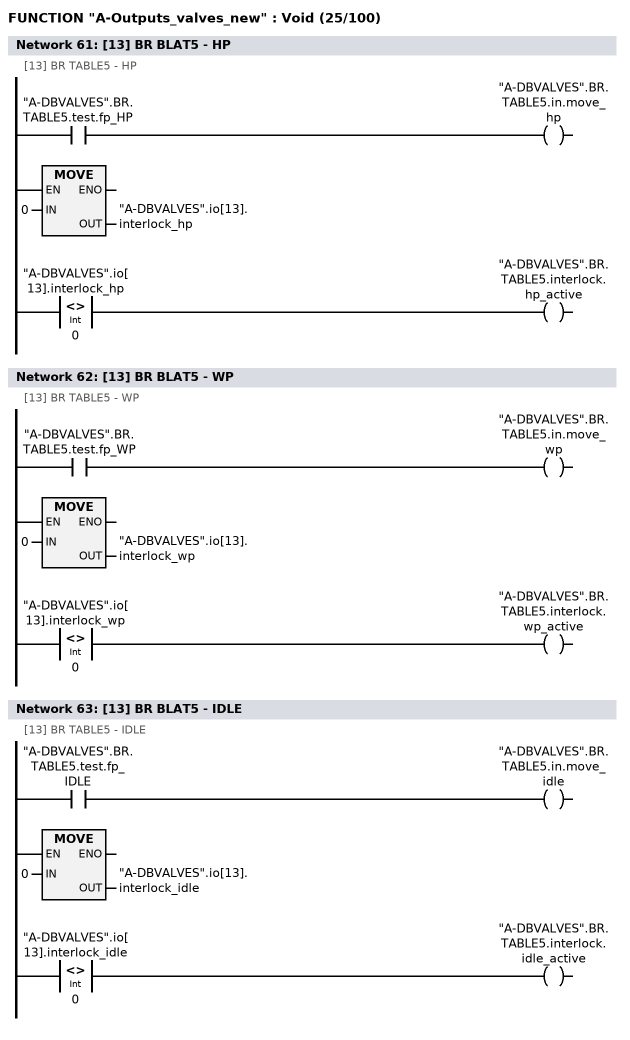
      O "A-DBVALVES".BR.TABLE5.test.fp_HP;
//    O     "A-Flags".STATION.IN_HP_STEP
      = "A-DBVALVES".BR.TABLE5.in.move_hp;

// Interlock hp
      L 0;
      T "A-DBVALVES".io[13].interlock_hp;

//{INTERLOCK_HP13}

      A(;
      L "A-DBVALVES".io[13].interlock_hp;
      L 0;
      <>I;
      );
      = "A-DBVALVES".BR.TABLE5.interlock.hp_active;
NETWORK
TITLE = [13] BR BLAT5 - WP
//[13] BR TABLE5 - WP
      O "A-DBVALVES".BR.TABLE5.test.fp_WP;
      = "A-DBVALVES".BR.TABLE5.in.move_wp;

// Interlock wp
      L 0;
      T "A-DBVALVES".io[13].interlock_wp;

//{INTERLOCK_WP13}

      A(;
      L "A-DBVALVES".io[13].interlock_wp;
      L 0;
      <>I;
      );
      = "A-DBVALVES".BR.TABLE5.interlock.wp_active;
NETWORK
TITLE = [13] BR BLAT5 - IDLE
//[13] BR TABLE5 - IDLE
      O "A-DBVALVES".BR.TABLE5.test.fp_IDLE;
      = "A-DBVALVES".BR.TABLE5.in.move_idle;

// Interlock idle
      L 0;
      T "A-DBVALVES".io[13].interlock_idle;

//{INTERLOCK_IDLE13}

      A(;
      L "A-DBVALVES".io[13].interlock_idle;
      L 0;
      <>I;
      );
      = "A-DBVALVES".BR.TABLE5.interlock.idle_active;
NETWORK
TITLE = [13] BR BLAT5
//[13] BR TABLE5
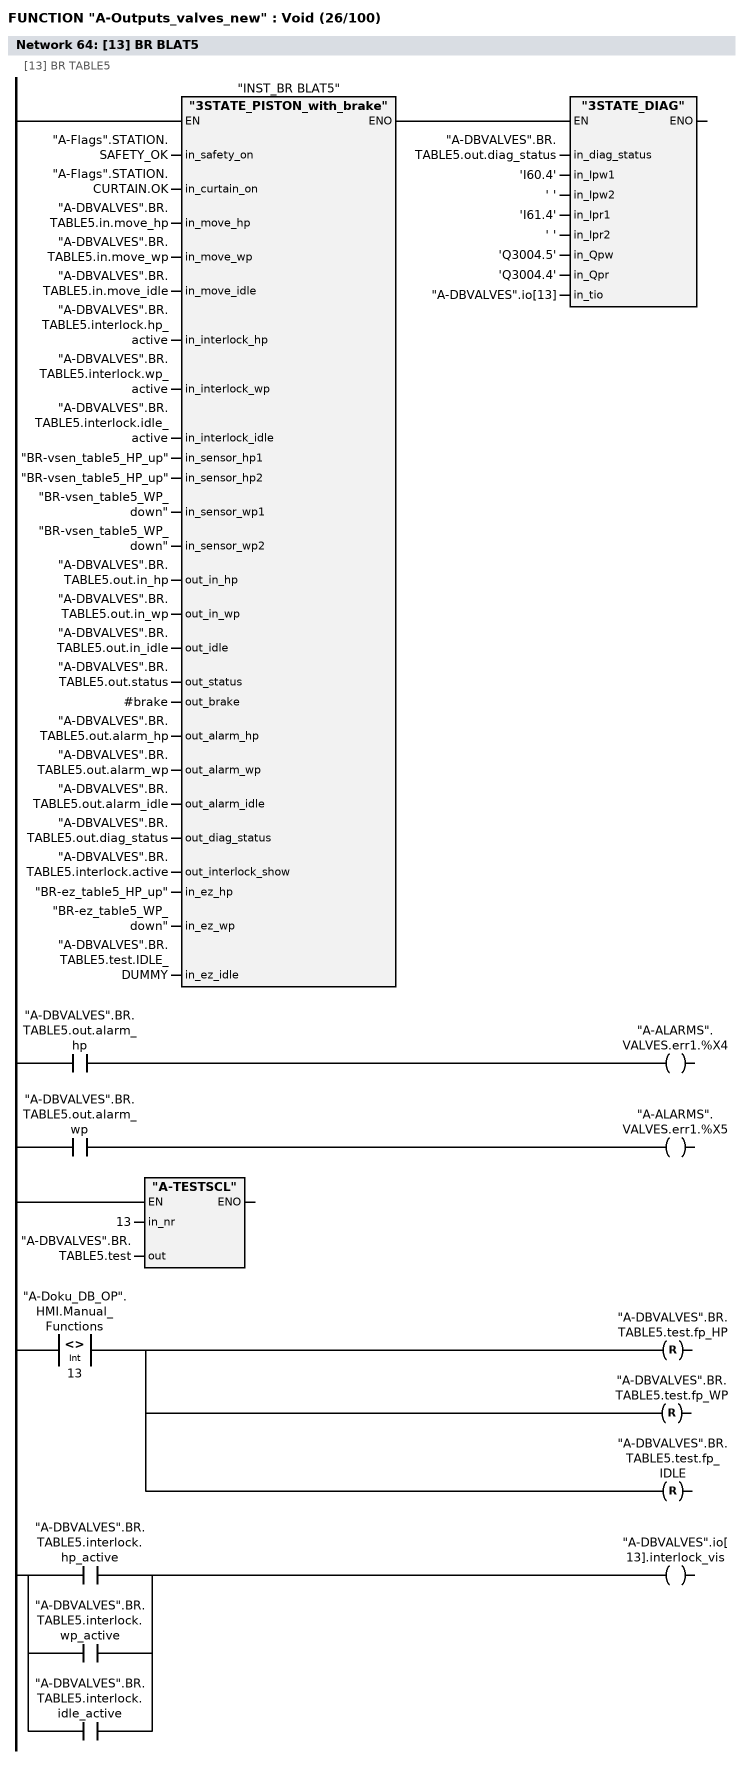
      CALL "3STATE_PISTON_with_brake", "INST_BR BLAT5"
      (  in_safety_on                := "A-Flags".STATION.SAFETY_OK ,
         in_curtain_on               := "A-Flags".STATION.CURTAIN.OK ,
         in_move_hp                  := "A-DBVALVES".BR.TABLE5.in.move_hp ,
         in_move_wp                  := "A-DBVALVES".BR.TABLE5.in.move_wp ,
         in_move_idle                := "A-DBVALVES".BR.TABLE5.in.move_idle ,
         in_interlock_hp             := "A-DBVALVES".BR.TABLE5.interlock.hp_active ,
         in_interlock_wp             := "A-DBVALVES".BR.TABLE5.interlock.wp_active ,
         in_interlock_idle           := "A-DBVALVES".BR.TABLE5.interlock.idle_active ,
         in_sensor_hp1               := "BR-vsen_table5_HP_up" ,
         in_sensor_hp2               := "BR-vsen_table5_HP_up" ,
         in_sensor_wp1               := "BR-vsen_table5_WP_down" ,
         in_sensor_wp2               := "BR-vsen_table5_WP_down" ,
         out_in_hp                   := "A-DBVALVES".BR.TABLE5.out.in_hp ,
         out_in_wp                   := "A-DBVALVES".BR.TABLE5.out.in_wp ,
         out_idle                    := "A-DBVALVES".BR.TABLE5.out.in_idle ,
         out_status                  := "A-DBVALVES".BR.TABLE5.out.status ,
         out_brake                   := #brake ,
         out_alarm_hp                := "A-DBVALVES".BR.TABLE5.out.alarm_hp ,
         out_alarm_wp                := "A-DBVALVES".BR.TABLE5.out.alarm_wp ,
         out_alarm_idle              := "A-DBVALVES".BR.TABLE5.out.alarm_idle ,
         out_diag_status             := "A-DBVALVES".BR.TABLE5.out.diag_status ,
         out_interlock_show          := "A-DBVALVES".BR.TABLE5.interlock.active ,
         in_ez_hp                    := "BR-ez_table5_HP_up" ,
         in_ez_wp                    := "BR-ez_table5_WP_down" ,
         in_ez_idle                  := "A-DBVALVES".BR.TABLE5.test.IDLE_DUMMY
      );

      CALL "3STATE_DIAG"
      (  in_diag_status              := "A-DBVALVES".BR.TABLE5.out.diag_status ,
         in_Ipw1                     := 'I60.4' ,
         in_Ipw2                     := ' ' ,
         in_Ipr1                     := 'I61.4' ,
         in_Ipr2                     := ' ' ,
         in_Qpw                      := 'Q3004.5' ,
         in_Qpr                      := 'Q3004.4' ,
         in_tio                      := "A-DBVALVES".io[13]
      );

      A "A-DBVALVES".BR.TABLE5.out.alarm_hp;
      = "A-ALARMS".VALVES.err1.%X4;

      A "A-DBVALVES".BR.TABLE5.out.alarm_wp;
      = "A-ALARMS".VALVES.err1.%X5;

      CALL "A-TESTSCL"
      (  in_nr                       := 13 ,
         out                         := "A-DBVALVES".BR.TABLE5.test
      );

      A(;
      L "A-Doku_DB_OP".HMI.Manual_Functions;
      L 13;
      <>I;
      );
      R "A-DBVALVES".BR.TABLE5.test.fp_HP;
      R "A-DBVALVES".BR.TABLE5.test.fp_WP;
      R "A-DBVALVES".BR.TABLE5.test.fp_IDLE;

      O "A-DBVALVES".BR.TABLE5.interlock.hp_active;
      O "A-DBVALVES".BR.TABLE5.interlock.wp_active;
      O "A-DBVALVES".BR.TABLE5.interlock.idle_active;
      = "A-DBVALVES".io[13].interlock_vis;
NETWORK
TITLE = -

NETWORK
TITLE = [14] BR BLAT_LEWY - HP
//[14] BR TABLE_LEFT - HP
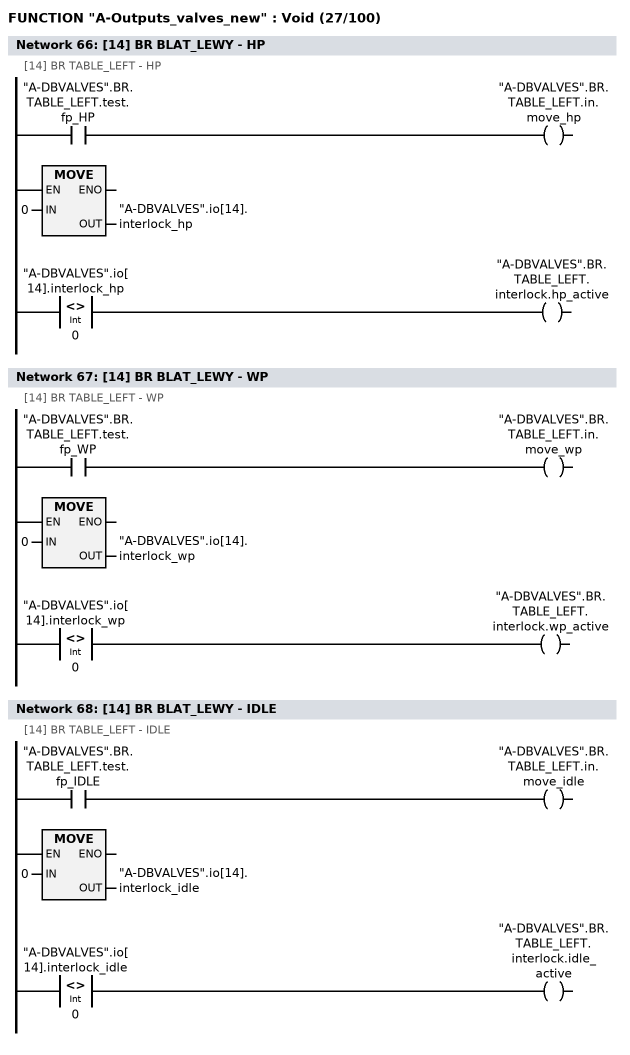
      O "A-DBVALVES".BR.TABLE_LEFT.test.fp_HP;
//    O     "A-Flags".STATION.IN_HP_STEP
      = "A-DBVALVES".BR.TABLE_LEFT.in.move_hp;

// Interlock hp
      L 0;
      T "A-DBVALVES".io[14].interlock_hp;

//{INTERLOCK_HP14}

      A(;
      L "A-DBVALVES".io[14].interlock_hp;
      L 0;
      <>I;
      );
      = "A-DBVALVES".BR.TABLE_LEFT.interlock.hp_active;
NETWORK
TITLE = [14] BR BLAT_LEWY - WP
//[14] BR TABLE_LEFT - WP
      O "A-DBVALVES".BR.TABLE_LEFT.test.fp_WP;
      = "A-DBVALVES".BR.TABLE_LEFT.in.move_wp;

// Interlock wp
      L 0;
      T "A-DBVALVES".io[14].interlock_wp;

//{INTERLOCK_WP14}

      A(;
      L "A-DBVALVES".io[14].interlock_wp;
      L 0;
      <>I;
      );
      = "A-DBVALVES".BR.TABLE_LEFT.interlock.wp_active;
NETWORK
TITLE = [14] BR BLAT_LEWY - IDLE
//[14] BR TABLE_LEFT - IDLE
      O "A-DBVALVES".BR.TABLE_LEFT.test.fp_IDLE;
      = "A-DBVALVES".BR.TABLE_LEFT.in.move_idle;

// Interlock idle
      L 0;
      T "A-DBVALVES".io[14].interlock_idle;

//{INTERLOCK_IDLE14}

      A(;
      L "A-DBVALVES".io[14].interlock_idle;
      L 0;
      <>I;
      );
      = "A-DBVALVES".BR.TABLE_LEFT.interlock.idle_active;
NETWORK
TITLE = [14] BR BLAT_LEWY
//[14] BR TABLE_LEFT
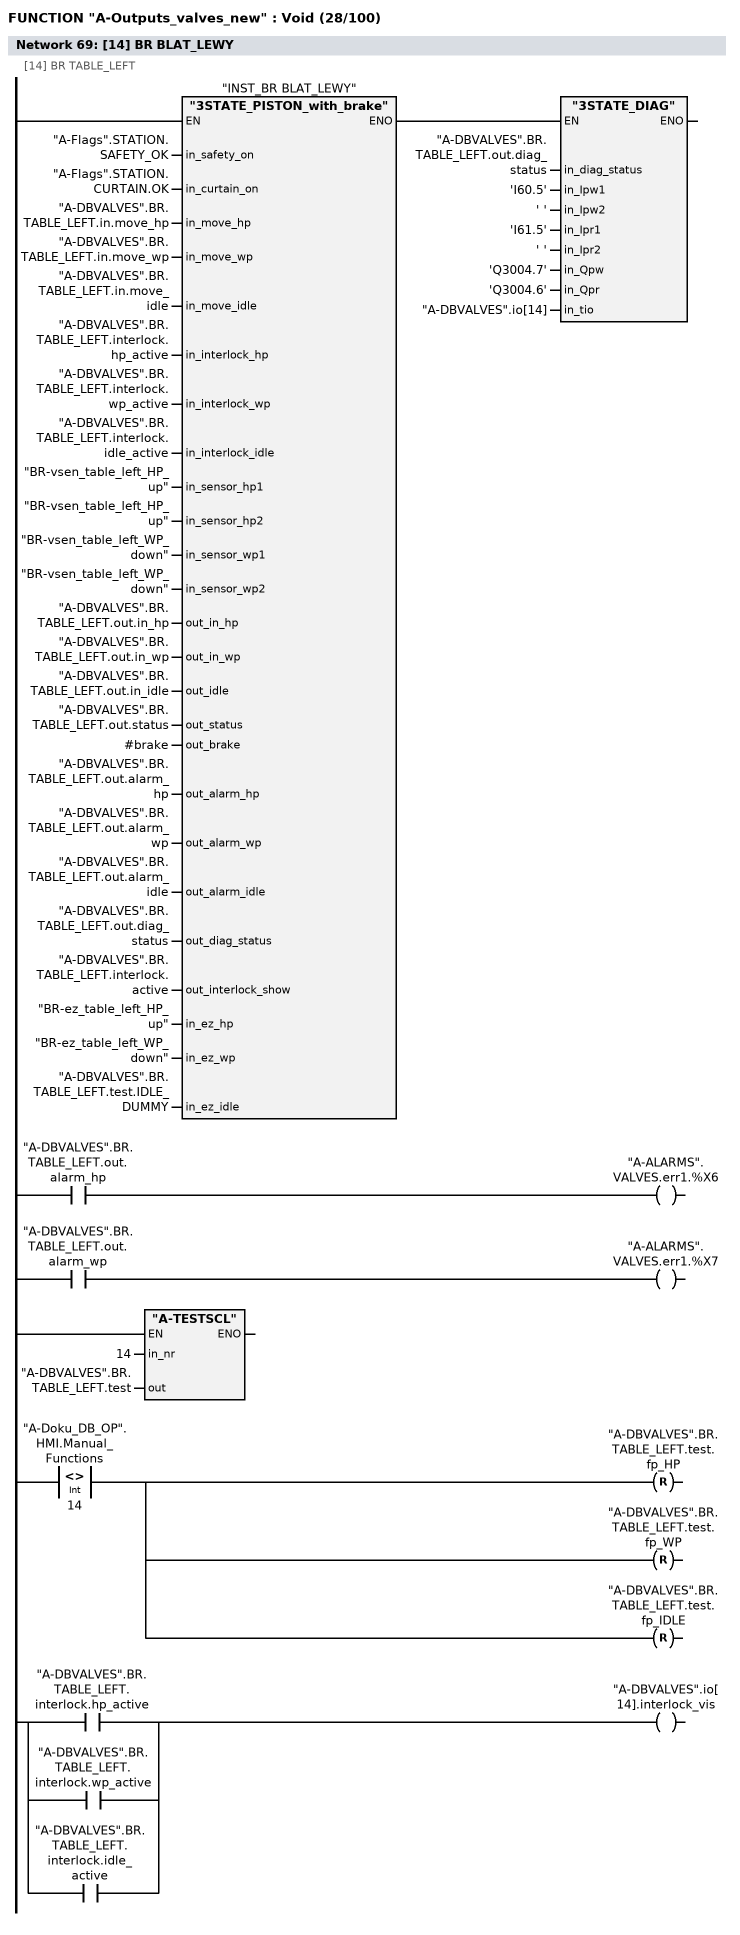
      CALL "3STATE_PISTON_with_brake", "INST_BR BLAT_LEWY"
      (  in_safety_on                := "A-Flags".STATION.SAFETY_OK ,
         in_curtain_on               := "A-Flags".STATION.CURTAIN.OK ,
         in_move_hp                  := "A-DBVALVES".BR.TABLE_LEFT.in.move_hp ,
         in_move_wp                  := "A-DBVALVES".BR.TABLE_LEFT.in.move_wp ,
         in_move_idle                := "A-DBVALVES".BR.TABLE_LEFT.in.move_idle ,
         in_interlock_hp             := "A-DBVALVES".BR.TABLE_LEFT.interlock.hp_active ,
         in_interlock_wp             := "A-DBVALVES".BR.TABLE_LEFT.interlock.wp_active ,
         in_interlock_idle           := "A-DBVALVES".BR.TABLE_LEFT.interlock.idle_active ,
         in_sensor_hp1               := "BR-vsen_table_left_HP_up" ,
         in_sensor_hp2               := "BR-vsen_table_left_HP_up" ,
         in_sensor_wp1               := "BR-vsen_table_left_WP_down" ,
         in_sensor_wp2               := "BR-vsen_table_left_WP_down" ,
         out_in_hp                   := "A-DBVALVES".BR.TABLE_LEFT.out.in_hp ,
         out_in_wp                   := "A-DBVALVES".BR.TABLE_LEFT.out.in_wp ,
         out_idle                    := "A-DBVALVES".BR.TABLE_LEFT.out.in_idle ,
         out_status                  := "A-DBVALVES".BR.TABLE_LEFT.out.status ,
         out_brake                   := #brake ,
         out_alarm_hp                := "A-DBVALVES".BR.TABLE_LEFT.out.alarm_hp ,
         out_alarm_wp                := "A-DBVALVES".BR.TABLE_LEFT.out.alarm_wp ,
         out_alarm_idle              := "A-DBVALVES".BR.TABLE_LEFT.out.alarm_idle ,
         out_diag_status             := "A-DBVALVES".BR.TABLE_LEFT.out.diag_status ,
         out_interlock_show          := "A-DBVALVES".BR.TABLE_LEFT.interlock.active ,
         in_ez_hp                    := "BR-ez_table_left_HP_up" ,
         in_ez_wp                    := "BR-ez_table_left_WP_down" ,
         in_ez_idle                  := "A-DBVALVES".BR.TABLE_LEFT.test.IDLE_DUMMY
      );

      CALL "3STATE_DIAG"
      (  in_diag_status              := "A-DBVALVES".BR.TABLE_LEFT.out.diag_status ,
         in_Ipw1                     := 'I60.5' ,
         in_Ipw2                     := ' ' ,
         in_Ipr1                     := 'I61.5' ,
         in_Ipr2                     := ' ' ,
         in_Qpw                      := 'Q3004.7' ,
         in_Qpr                      := 'Q3004.6' ,
         in_tio                      := "A-DBVALVES".io[14]
      );

      A "A-DBVALVES".BR.TABLE_LEFT.out.alarm_hp;
      = "A-ALARMS".VALVES.err1.%X6;

      A "A-DBVALVES".BR.TABLE_LEFT.out.alarm_wp;
      = "A-ALARMS".VALVES.err1.%X7;

      CALL "A-TESTSCL"
      (  in_nr                       := 14 ,
         out                         := "A-DBVALVES".BR.TABLE_LEFT.test
      );

      A(;
      L "A-Doku_DB_OP".HMI.Manual_Functions;
      L 14;
      <>I;
      );
      R "A-DBVALVES".BR.TABLE_LEFT.test.fp_HP;
      R "A-DBVALVES".BR.TABLE_LEFT.test.fp_WP;
      R "A-DBVALVES".BR.TABLE_LEFT.test.fp_IDLE;

      O "A-DBVALVES".BR.TABLE_LEFT.interlock.hp_active;
      O "A-DBVALVES".BR.TABLE_LEFT.interlock.wp_active;
      O "A-DBVALVES".BR.TABLE_LEFT.interlock.idle_active;
      = "A-DBVALVES".io[14].interlock_vis;
NETWORK
TITLE = -

NETWORK
TITLE = [15] BR BLAT_PRAWY - HP
//[15] BR TABLE_RIGHT - HP
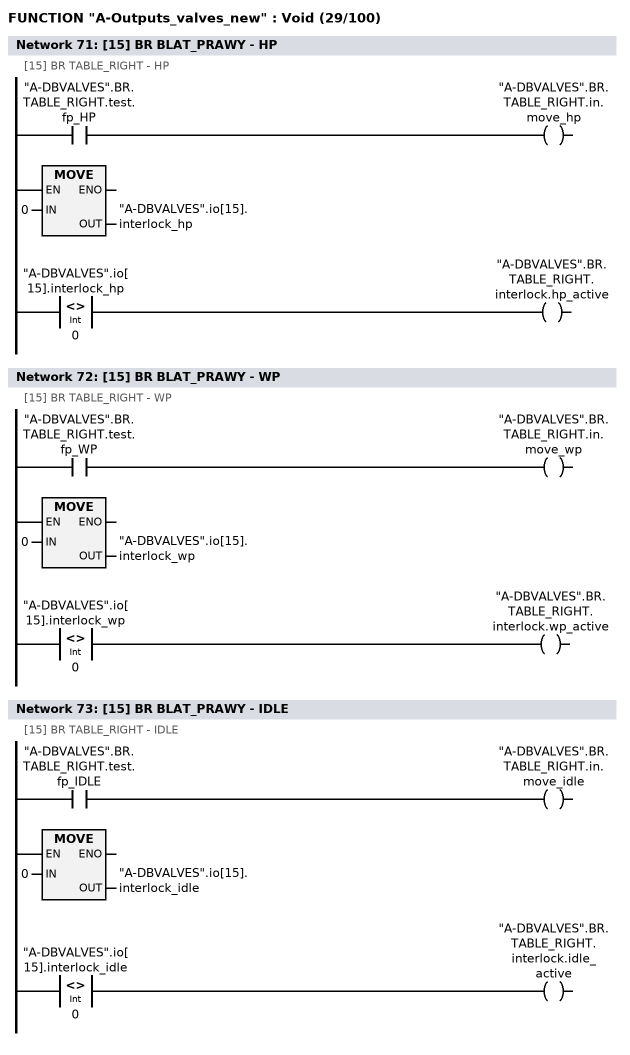
      O "A-DBVALVES".BR.TABLE_RIGHT.test.fp_HP;
//    O     "A-Flags".STATION.IN_HP_STEP
      = "A-DBVALVES".BR.TABLE_RIGHT.in.move_hp;

// Interlock hp
      L 0;
      T "A-DBVALVES".io[15].interlock_hp;

//{INTERLOCK_HP15}

      A(;
      L "A-DBVALVES".io[15].interlock_hp;
      L 0;
      <>I;
      );
      = "A-DBVALVES".BR.TABLE_RIGHT.interlock.hp_active;
NETWORK
TITLE = [15] BR BLAT_PRAWY - WP
//[15] BR TABLE_RIGHT - WP
      O "A-DBVALVES".BR.TABLE_RIGHT.test.fp_WP;
      = "A-DBVALVES".BR.TABLE_RIGHT.in.move_wp;

// Interlock wp
      L 0;
      T "A-DBVALVES".io[15].interlock_wp;

//{INTERLOCK_WP15}

      A(;
      L "A-DBVALVES".io[15].interlock_wp;
      L 0;
      <>I;
      );
      = "A-DBVALVES".BR.TABLE_RIGHT.interlock.wp_active;
NETWORK
TITLE = [15] BR BLAT_PRAWY - IDLE
//[15] BR TABLE_RIGHT - IDLE
      O "A-DBVALVES".BR.TABLE_RIGHT.test.fp_IDLE;
      = "A-DBVALVES".BR.TABLE_RIGHT.in.move_idle;

// Interlock idle
      L 0;
      T "A-DBVALVES".io[15].interlock_idle;

//{INTERLOCK_IDLE15}

      A(;
      L "A-DBVALVES".io[15].interlock_idle;
      L 0;
      <>I;
      );
      = "A-DBVALVES".BR.TABLE_RIGHT.interlock.idle_active;
NETWORK
TITLE = [15] BR BLAT_PRAWY
//[15] BR TABLE_RIGHT
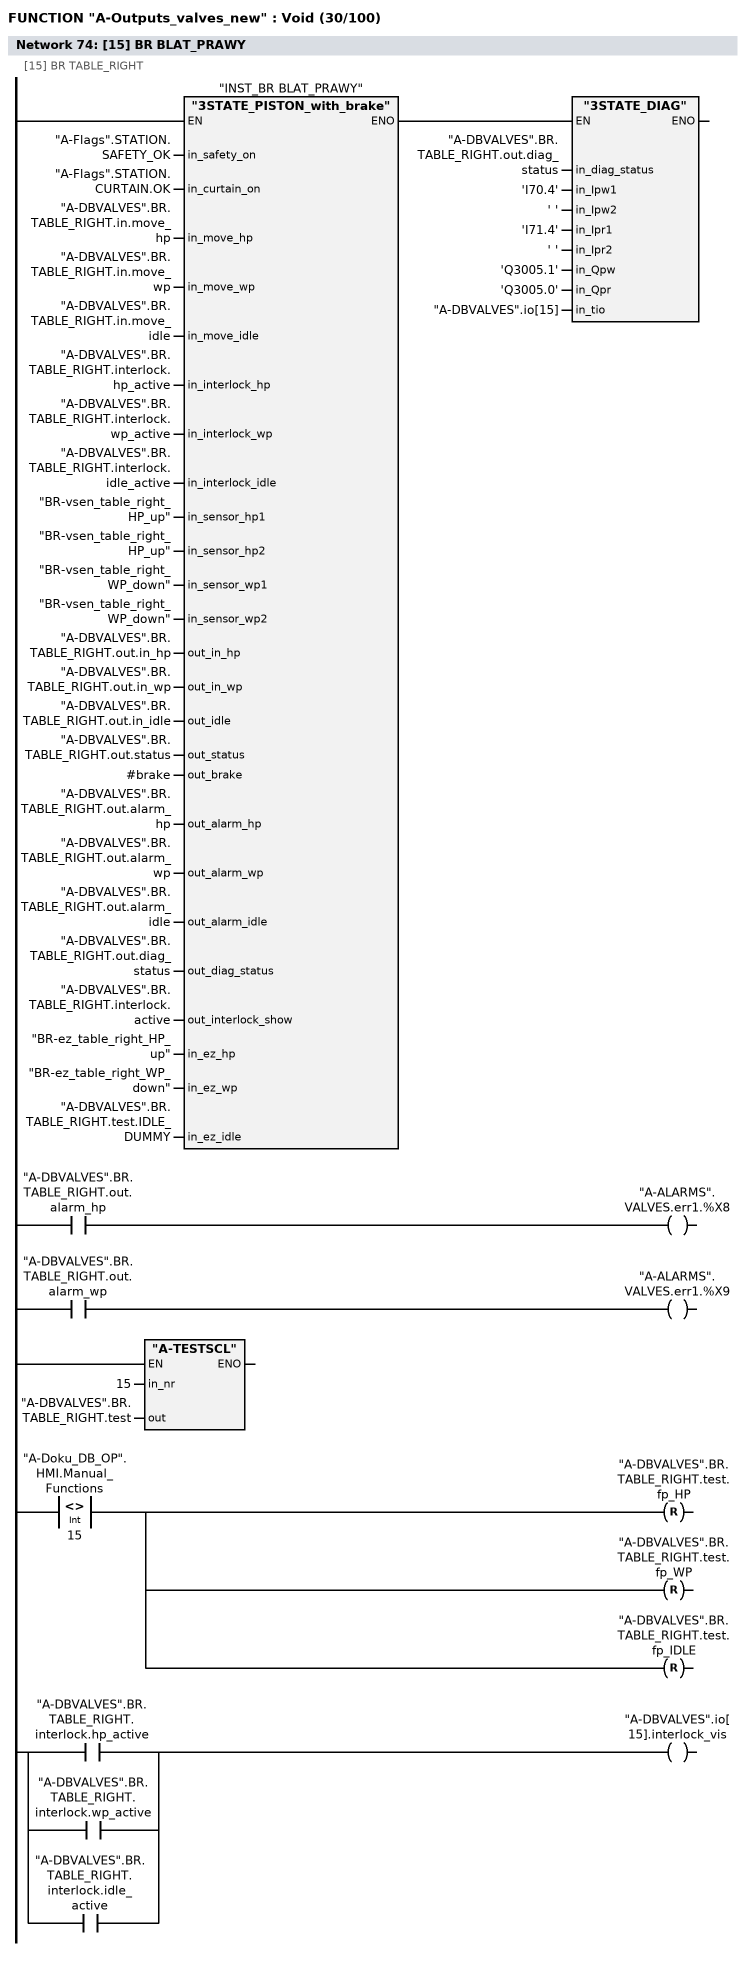
      CALL "3STATE_PISTON_with_brake", "INST_BR BLAT_PRAWY"
      (  in_safety_on                := "A-Flags".STATION.SAFETY_OK ,
         in_curtain_on               := "A-Flags".STATION.CURTAIN.OK ,
         in_move_hp                  := "A-DBVALVES".BR.TABLE_RIGHT.in.move_hp ,
         in_move_wp                  := "A-DBVALVES".BR.TABLE_RIGHT.in.move_wp ,
         in_move_idle                := "A-DBVALVES".BR.TABLE_RIGHT.in.move_idle ,
         in_interlock_hp             := "A-DBVALVES".BR.TABLE_RIGHT.interlock.hp_active ,
         in_interlock_wp             := "A-DBVALVES".BR.TABLE_RIGHT.interlock.wp_active ,
         in_interlock_idle           := "A-DBVALVES".BR.TABLE_RIGHT.interlock.idle_active ,
         in_sensor_hp1               := "BR-vsen_table_right_HP_up" ,
         in_sensor_hp2               := "BR-vsen_table_right_HP_up" ,
         in_sensor_wp1               := "BR-vsen_table_right_WP_down" ,
         in_sensor_wp2               := "BR-vsen_table_right_WP_down" ,
         out_in_hp                   := "A-DBVALVES".BR.TABLE_RIGHT.out.in_hp ,
         out_in_wp                   := "A-DBVALVES".BR.TABLE_RIGHT.out.in_wp ,
         out_idle                    := "A-DBVALVES".BR.TABLE_RIGHT.out.in_idle ,
         out_status                  := "A-DBVALVES".BR.TABLE_RIGHT.out.status ,
         out_brake                   := #brake ,
         out_alarm_hp                := "A-DBVALVES".BR.TABLE_RIGHT.out.alarm_hp ,
         out_alarm_wp                := "A-DBVALVES".BR.TABLE_RIGHT.out.alarm_wp ,
         out_alarm_idle              := "A-DBVALVES".BR.TABLE_RIGHT.out.alarm_idle ,
         out_diag_status             := "A-DBVALVES".BR.TABLE_RIGHT.out.diag_status ,
         out_interlock_show          := "A-DBVALVES".BR.TABLE_RIGHT.interlock.active ,
         in_ez_hp                    := "BR-ez_table_right_HP_up" ,
         in_ez_wp                    := "BR-ez_table_right_WP_down" ,
         in_ez_idle                  := "A-DBVALVES".BR.TABLE_RIGHT.test.IDLE_DUMMY
      );

      CALL "3STATE_DIAG"
      (  in_diag_status              := "A-DBVALVES".BR.TABLE_RIGHT.out.diag_status ,
         in_Ipw1                     := 'I70.4' ,
         in_Ipw2                     := ' ' ,
         in_Ipr1                     := 'I71.4' ,
         in_Ipr2                     := ' ' ,
         in_Qpw                      := 'Q3005.1' ,
         in_Qpr                      := 'Q3005.0' ,
         in_tio                      := "A-DBVALVES".io[15]
      );

      A "A-DBVALVES".BR.TABLE_RIGHT.out.alarm_hp;
      = "A-ALARMS".VALVES.err1.%X8;

      A "A-DBVALVES".BR.TABLE_RIGHT.out.alarm_wp;
      = "A-ALARMS".VALVES.err1.%X9;

      CALL "A-TESTSCL"
      (  in_nr                       := 15 ,
         out                         := "A-DBVALVES".BR.TABLE_RIGHT.test
      );

      A(;
      L "A-Doku_DB_OP".HMI.Manual_Functions;
      L 15;
      <>I;
      );
      R "A-DBVALVES".BR.TABLE_RIGHT.test.fp_HP;
      R "A-DBVALVES".BR.TABLE_RIGHT.test.fp_WP;
      R "A-DBVALVES".BR.TABLE_RIGHT.test.fp_IDLE;

      O "A-DBVALVES".BR.TABLE_RIGHT.interlock.hp_active;
      O "A-DBVALVES".BR.TABLE_RIGHT.interlock.wp_active;
      O "A-DBVALVES".BR.TABLE_RIGHT.interlock.idle_active;
      = "A-DBVALVES".io[15].interlock_vis;
NETWORK
TITLE = -

NETWORK
TITLE = [16] ST1 STACJA_PRZESUW - HP
//[16] ST1 STATION_MOVEMENT - HP
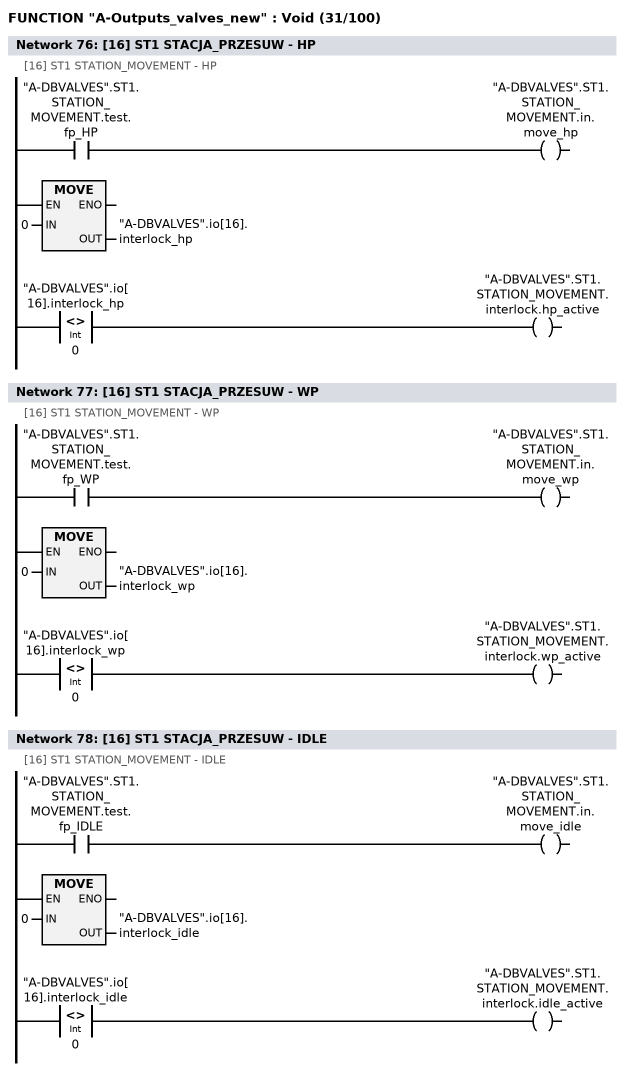
      O "A-DBVALVES".ST1.STATION_MOVEMENT.test.fp_HP;
//    O     "A-Flags".STATION.IN_HP_STEP
      = "A-DBVALVES".ST1.STATION_MOVEMENT.in.move_hp;

// Interlock hp
      L 0;
      T "A-DBVALVES".io[16].interlock_hp;

//{INTERLOCK_HP16}

      A(;
      L "A-DBVALVES".io[16].interlock_hp;
      L 0;
      <>I;
      );
      = "A-DBVALVES".ST1.STATION_MOVEMENT.interlock.hp_active;
NETWORK
TITLE = [16] ST1 STACJA_PRZESUW - WP
//[16] ST1 STATION_MOVEMENT - WP
      O "A-DBVALVES".ST1.STATION_MOVEMENT.test.fp_WP;
      = "A-DBVALVES".ST1.STATION_MOVEMENT.in.move_wp;

// Interlock wp
      L 0;
      T "A-DBVALVES".io[16].interlock_wp;

//{INTERLOCK_WP16}

      A(;
      L "A-DBVALVES".io[16].interlock_wp;
      L 0;
      <>I;
      );
      = "A-DBVALVES".ST1.STATION_MOVEMENT.interlock.wp_active;
NETWORK
TITLE = [16] ST1 STACJA_PRZESUW - IDLE
//[16] ST1 STATION_MOVEMENT - IDLE
      O "A-DBVALVES".ST1.STATION_MOVEMENT.test.fp_IDLE;
      = "A-DBVALVES".ST1.STATION_MOVEMENT.in.move_idle;

// Interlock idle
      L 0;
      T "A-DBVALVES".io[16].interlock_idle;

//{INTERLOCK_IDLE16}

      A(;
      L "A-DBVALVES".io[16].interlock_idle;
      L 0;
      <>I;
      );
      = "A-DBVALVES".ST1.STATION_MOVEMENT.interlock.idle_active;
NETWORK
TITLE = [16] ST1 STACJA_PRZESUW
//[16] ST1 STATION_MOVEMENT
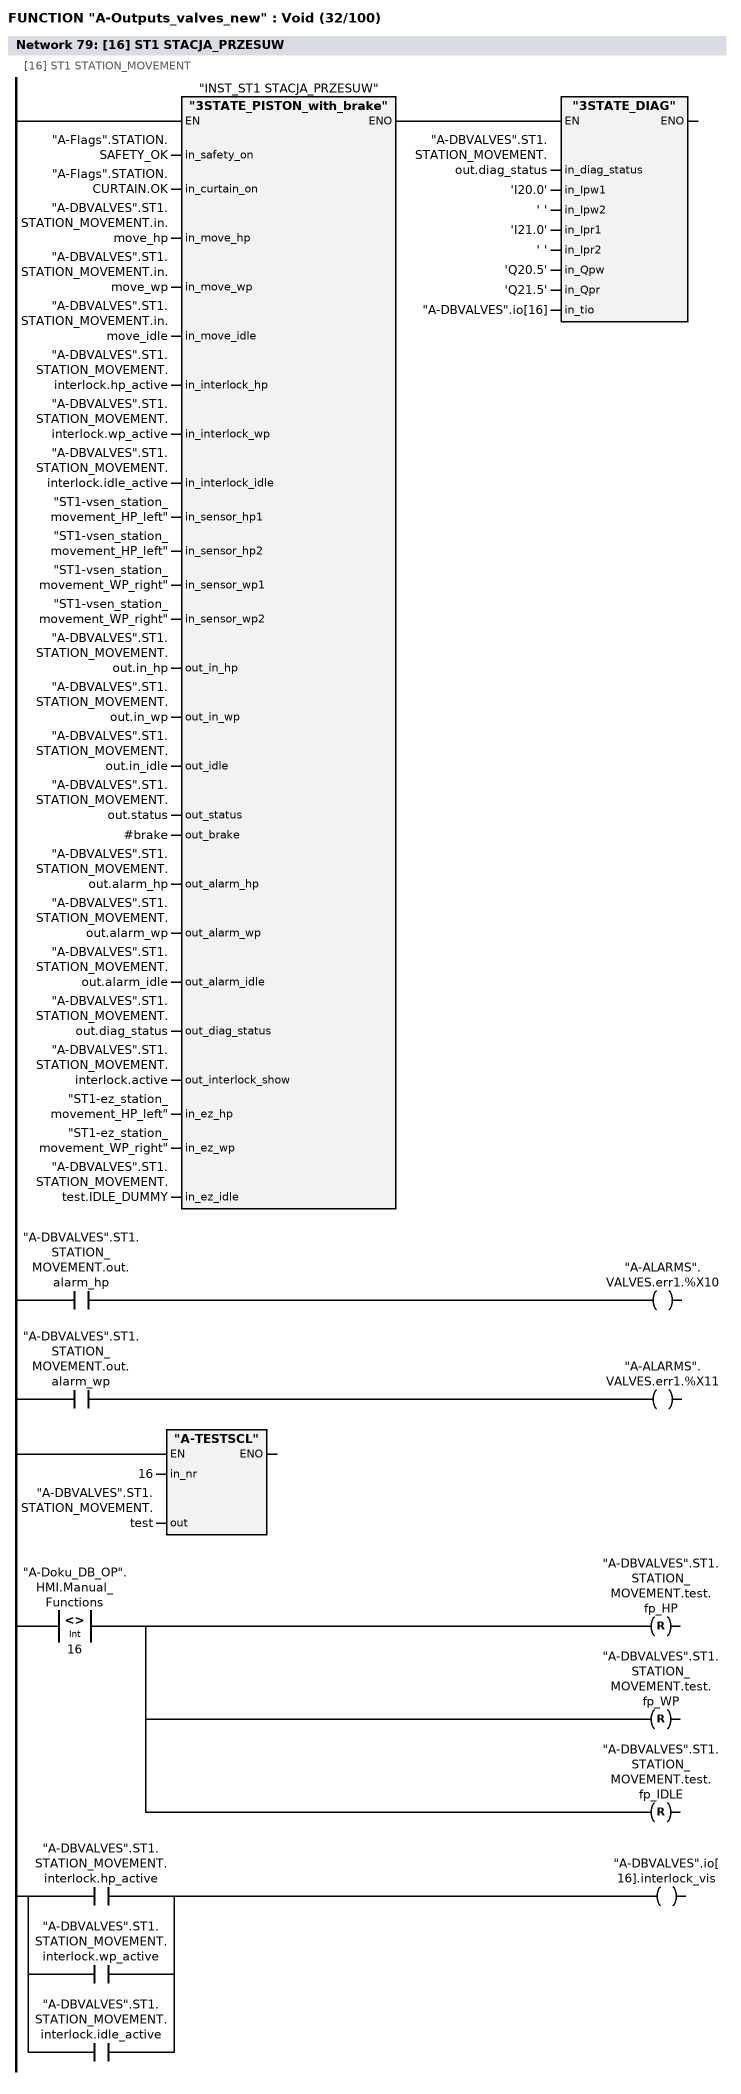
      CALL "3STATE_PISTON_with_brake", "INST_ST1 STACJA_PRZESUW"
      (  in_safety_on                := "A-Flags".STATION.SAFETY_OK ,
         in_curtain_on               := "A-Flags".STATION.CURTAIN.OK ,
         in_move_hp                  := "A-DBVALVES".ST1.STATION_MOVEMENT.in.move_hp ,
         in_move_wp                  := "A-DBVALVES".ST1.STATION_MOVEMENT.in.move_wp ,
         in_move_idle                := "A-DBVALVES".ST1.STATION_MOVEMENT.in.move_idle ,
         in_interlock_hp             := "A-DBVALVES".ST1.STATION_MOVEMENT.interlock.hp_active ,
         in_interlock_wp             := "A-DBVALVES".ST1.STATION_MOVEMENT.interlock.wp_active ,
         in_interlock_idle           := "A-DBVALVES".ST1.STATION_MOVEMENT.interlock.idle_active ,
         in_sensor_hp1               := "ST1-vsen_station_movement_HP_left" ,
         in_sensor_hp2               := "ST1-vsen_station_movement_HP_left" ,
         in_sensor_wp1               := "ST1-vsen_station_movement_WP_right" ,
         in_sensor_wp2               := "ST1-vsen_station_movement_WP_right" ,
         out_in_hp                   := "A-DBVALVES".ST1.STATION_MOVEMENT.out.in_hp ,
         out_in_wp                   := "A-DBVALVES".ST1.STATION_MOVEMENT.out.in_wp ,
         out_idle                    := "A-DBVALVES".ST1.STATION_MOVEMENT.out.in_idle ,
         out_status                  := "A-DBVALVES".ST1.STATION_MOVEMENT.out.status ,
         out_brake                   := #brake ,
         out_alarm_hp                := "A-DBVALVES".ST1.STATION_MOVEMENT.out.alarm_hp ,
         out_alarm_wp                := "A-DBVALVES".ST1.STATION_MOVEMENT.out.alarm_wp ,
         out_alarm_idle              := "A-DBVALVES".ST1.STATION_MOVEMENT.out.alarm_idle ,
         out_diag_status             := "A-DBVALVES".ST1.STATION_MOVEMENT.out.diag_status ,
         out_interlock_show          := "A-DBVALVES".ST1.STATION_MOVEMENT.interlock.active ,
         in_ez_hp                    := "ST1-ez_station_movement_HP_left" ,
         in_ez_wp                    := "ST1-ez_station_movement_WP_right" ,
         in_ez_idle                  := "A-DBVALVES".ST1.STATION_MOVEMENT.test.IDLE_DUMMY
      );

      CALL "3STATE_DIAG"
      (  in_diag_status              := "A-DBVALVES".ST1.STATION_MOVEMENT.out.diag_status ,
         in_Ipw1                     := 'I20.0' ,
         in_Ipw2                     := ' ' ,
         in_Ipr1                     := 'I21.0' ,
         in_Ipr2                     := ' ' ,
         in_Qpw                      := 'Q20.5' ,
         in_Qpr                      := 'Q21.5' ,
         in_tio                      := "A-DBVALVES".io[16]
      );

      A "A-DBVALVES".ST1.STATION_MOVEMENT.out.alarm_hp;
      = "A-ALARMS".VALVES.err1.%X10;

      A "A-DBVALVES".ST1.STATION_MOVEMENT.out.alarm_wp;
      = "A-ALARMS".VALVES.err1.%X11;

      CALL "A-TESTSCL"
      (  in_nr                       := 16 ,
         out                         := "A-DBVALVES".ST1.STATION_MOVEMENT.test
      );

      A(;
      L "A-Doku_DB_OP".HMI.Manual_Functions;
      L 16;
      <>I;
      );
      R "A-DBVALVES".ST1.STATION_MOVEMENT.test.fp_HP;
      R "A-DBVALVES".ST1.STATION_MOVEMENT.test.fp_WP;
      R "A-DBVALVES".ST1.STATION_MOVEMENT.test.fp_IDLE;

      O "A-DBVALVES".ST1.STATION_MOVEMENT.interlock.hp_active;
      O "A-DBVALVES".ST1.STATION_MOVEMENT.interlock.wp_active;
      O "A-DBVALVES".ST1.STATION_MOVEMENT.interlock.idle_active;
      = "A-DBVALVES".io[16].interlock_vis;
NETWORK
TITLE = -

NETWORK
TITLE = [17] ST1 MIECZ_WYSUW - HP
//[17] ST1 SWORD_SLIDE_OUT - HP
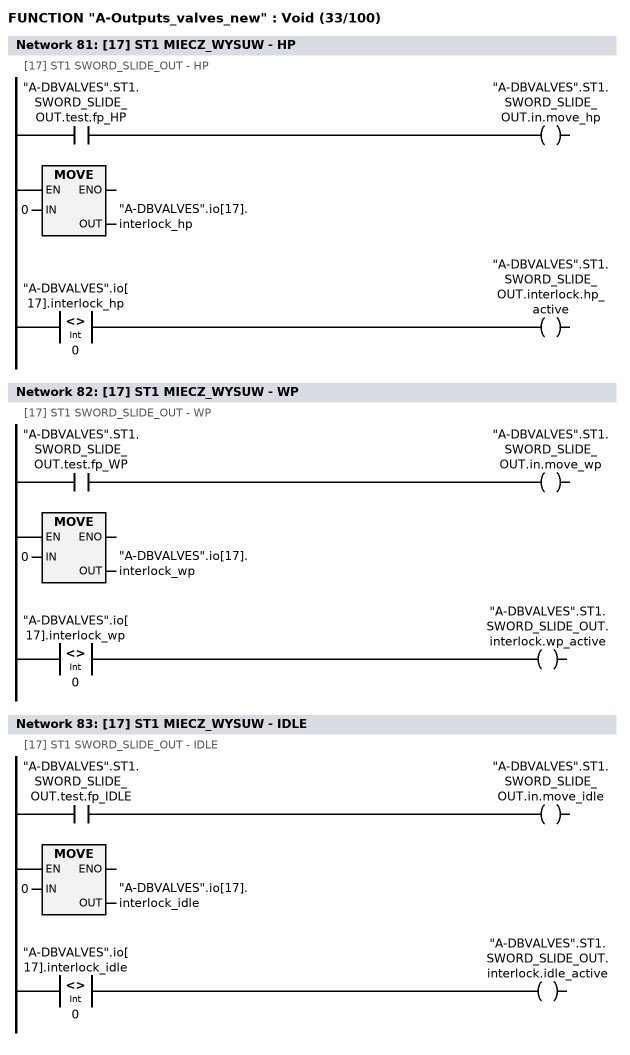
      O "A-DBVALVES".ST1.SWORD_SLIDE_OUT.test.fp_HP;
//    O     "A-Flags".STATION.IN_HP_STEP
      = "A-DBVALVES".ST1.SWORD_SLIDE_OUT.in.move_hp;

// Interlock hp
      L 0;
      T "A-DBVALVES".io[17].interlock_hp;

//{INTERLOCK_HP17}

      A(;
      L "A-DBVALVES".io[17].interlock_hp;
      L 0;
      <>I;
      );
      = "A-DBVALVES".ST1.SWORD_SLIDE_OUT.interlock.hp_active;
NETWORK
TITLE = [17] ST1 MIECZ_WYSUW - WP
//[17] ST1 SWORD_SLIDE_OUT - WP
      O "A-DBVALVES".ST1.SWORD_SLIDE_OUT.test.fp_WP;
      = "A-DBVALVES".ST1.SWORD_SLIDE_OUT.in.move_wp;

// Interlock wp
      L 0;
      T "A-DBVALVES".io[17].interlock_wp;

//{INTERLOCK_WP17}

      A(;
      L "A-DBVALVES".io[17].interlock_wp;
      L 0;
      <>I;
      );
      = "A-DBVALVES".ST1.SWORD_SLIDE_OUT.interlock.wp_active;
NETWORK
TITLE = [17] ST1 MIECZ_WYSUW - IDLE
//[17] ST1 SWORD_SLIDE_OUT - IDLE
      O "A-DBVALVES".ST1.SWORD_SLIDE_OUT.test.fp_IDLE;
      = "A-DBVALVES".ST1.SWORD_SLIDE_OUT.in.move_idle;

// Interlock idle
      L 0;
      T "A-DBVALVES".io[17].interlock_idle;

//{INTERLOCK_IDLE17}

      A(;
      L "A-DBVALVES".io[17].interlock_idle;
      L 0;
      <>I;
      );
      = "A-DBVALVES".ST1.SWORD_SLIDE_OUT.interlock.idle_active;
NETWORK
TITLE = [17] ST1 MIECZ_WYSUW
//[17] ST1 SWORD_SLIDE_OUT
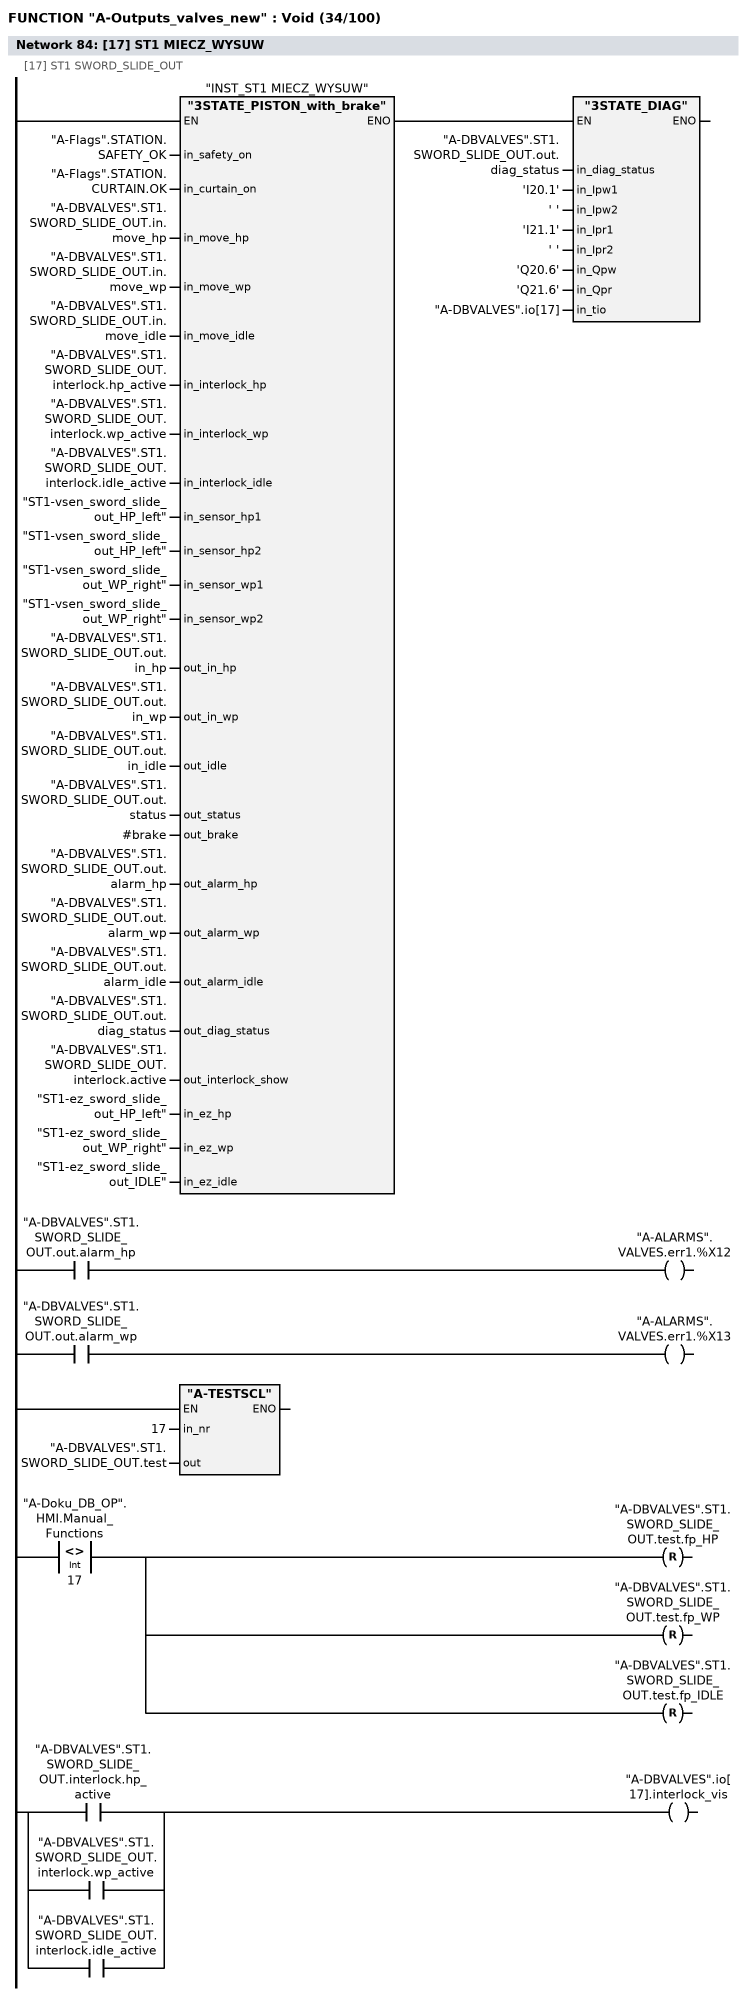
      CALL "3STATE_PISTON_with_brake", "INST_ST1 MIECZ_WYSUW"
      (  in_safety_on                := "A-Flags".STATION.SAFETY_OK ,
         in_curtain_on               := "A-Flags".STATION.CURTAIN.OK ,
         in_move_hp                  := "A-DBVALVES".ST1.SWORD_SLIDE_OUT.in.move_hp ,
         in_move_wp                  := "A-DBVALVES".ST1.SWORD_SLIDE_OUT.in.move_wp ,
         in_move_idle                := "A-DBVALVES".ST1.SWORD_SLIDE_OUT.in.move_idle ,
         in_interlock_hp             := "A-DBVALVES".ST1.SWORD_SLIDE_OUT.interlock.hp_active ,
         in_interlock_wp             := "A-DBVALVES".ST1.SWORD_SLIDE_OUT.interlock.wp_active ,
         in_interlock_idle           := "A-DBVALVES".ST1.SWORD_SLIDE_OUT.interlock.idle_active ,
         in_sensor_hp1               := "ST1-vsen_sword_slide_out_HP_left" ,
         in_sensor_hp2               := "ST1-vsen_sword_slide_out_HP_left" ,
         in_sensor_wp1               := "ST1-vsen_sword_slide_out_WP_right" ,
         in_sensor_wp2               := "ST1-vsen_sword_slide_out_WP_right" ,
         out_in_hp                   := "A-DBVALVES".ST1.SWORD_SLIDE_OUT.out.in_hp ,
         out_in_wp                   := "A-DBVALVES".ST1.SWORD_SLIDE_OUT.out.in_wp ,
         out_idle                    := "A-DBVALVES".ST1.SWORD_SLIDE_OUT.out.in_idle ,
         out_status                  := "A-DBVALVES".ST1.SWORD_SLIDE_OUT.out.status ,
         out_brake                   := #brake ,
         out_alarm_hp                := "A-DBVALVES".ST1.SWORD_SLIDE_OUT.out.alarm_hp ,
         out_alarm_wp                := "A-DBVALVES".ST1.SWORD_SLIDE_OUT.out.alarm_wp ,
         out_alarm_idle              := "A-DBVALVES".ST1.SWORD_SLIDE_OUT.out.alarm_idle ,
         out_diag_status             := "A-DBVALVES".ST1.SWORD_SLIDE_OUT.out.diag_status ,
         out_interlock_show          := "A-DBVALVES".ST1.SWORD_SLIDE_OUT.interlock.active ,
         in_ez_hp                    := "ST1-ez_sword_slide_out_HP_left" ,
         in_ez_wp                    := "ST1-ez_sword_slide_out_WP_right" ,
         in_ez_idle                  := "ST1-ez_sword_slide_out_IDLE"
      );

      CALL "3STATE_DIAG"
      (  in_diag_status              := "A-DBVALVES".ST1.SWORD_SLIDE_OUT.out.diag_status ,
         in_Ipw1                     := 'I20.1' ,
         in_Ipw2                     := ' ' ,
         in_Ipr1                     := 'I21.1' ,
         in_Ipr2                     := ' ' ,
         in_Qpw                      := 'Q20.6' ,
         in_Qpr                      := 'Q21.6' ,
         in_tio                      := "A-DBVALVES".io[17]
      );

      A "A-DBVALVES".ST1.SWORD_SLIDE_OUT.out.alarm_hp;
      = "A-ALARMS".VALVES.err1.%X12;

      A "A-DBVALVES".ST1.SWORD_SLIDE_OUT.out.alarm_wp;
      = "A-ALARMS".VALVES.err1.%X13;

      CALL "A-TESTSCL"
      (  in_nr                       := 17 ,
         out                         := "A-DBVALVES".ST1.SWORD_SLIDE_OUT.test
      );

      A(;
      L "A-Doku_DB_OP".HMI.Manual_Functions;
      L 17;
      <>I;
      );
      R "A-DBVALVES".ST1.SWORD_SLIDE_OUT.test.fp_HP;
      R "A-DBVALVES".ST1.SWORD_SLIDE_OUT.test.fp_WP;
      R "A-DBVALVES".ST1.SWORD_SLIDE_OUT.test.fp_IDLE;

      O "A-DBVALVES".ST1.SWORD_SLIDE_OUT.interlock.hp_active;
      O "A-DBVALVES".ST1.SWORD_SLIDE_OUT.interlock.wp_active;
      O "A-DBVALVES".ST1.SWORD_SLIDE_OUT.interlock.idle_active;
      = "A-DBVALVES".io[17].interlock_vis;
NETWORK
TITLE = -

NETWORK
TITLE = [18] ST1 MIECZ - HP
//[18] ST1 SWORD - HP
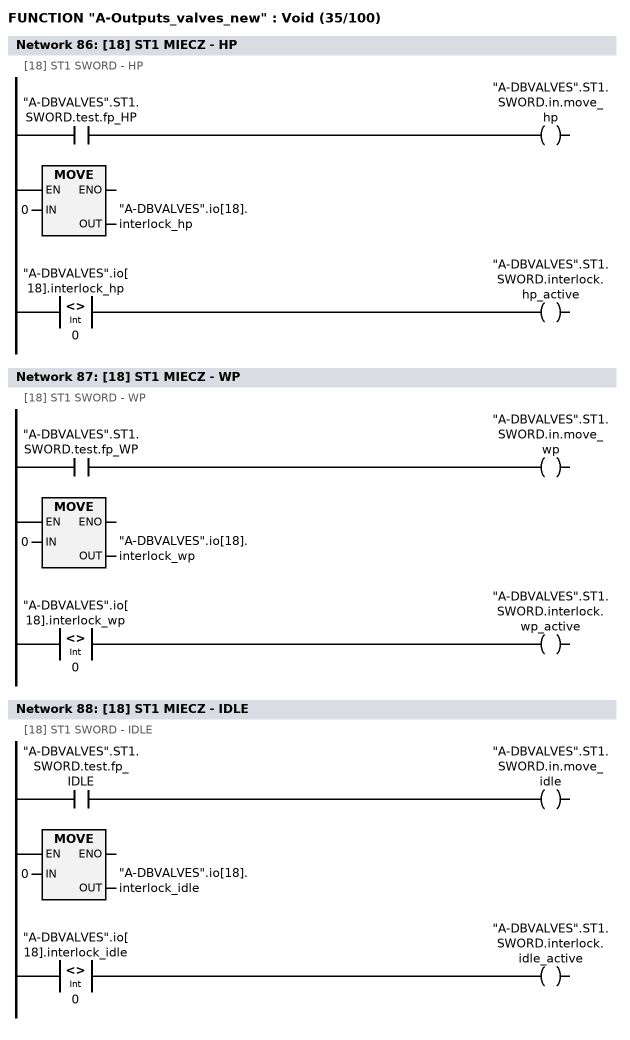
      O "A-DBVALVES".ST1.SWORD.test.fp_HP;
//    O     "A-Flags".STATION.IN_HP_STEP
      = "A-DBVALVES".ST1.SWORD.in.move_hp;

// Interlock hp
      L 0;
      T "A-DBVALVES".io[18].interlock_hp;

//{INTERLOCK_HP18}

      A(;
      L "A-DBVALVES".io[18].interlock_hp;
      L 0;
      <>I;
      );
      = "A-DBVALVES".ST1.SWORD.interlock.hp_active;
NETWORK
TITLE = [18] ST1 MIECZ - WP
//[18] ST1 SWORD - WP
      O "A-DBVALVES".ST1.SWORD.test.fp_WP;
      = "A-DBVALVES".ST1.SWORD.in.move_wp;

// Interlock wp
      L 0;
      T "A-DBVALVES".io[18].interlock_wp;

//{INTERLOCK_WP18}

      A(;
      L "A-DBVALVES".io[18].interlock_wp;
      L 0;
      <>I;
      );
      = "A-DBVALVES".ST1.SWORD.interlock.wp_active;
NETWORK
TITLE = [18] ST1 MIECZ - IDLE
//[18] ST1 SWORD - IDLE
      O "A-DBVALVES".ST1.SWORD.test.fp_IDLE;
      = "A-DBVALVES".ST1.SWORD.in.move_idle;

// Interlock idle
      L 0;
      T "A-DBVALVES".io[18].interlock_idle;

//{INTERLOCK_IDLE18}

      A(;
      L "A-DBVALVES".io[18].interlock_idle;
      L 0;
      <>I;
      );
      = "A-DBVALVES".ST1.SWORD.interlock.idle_active;
NETWORK
TITLE = [18] ST1 MIECZ
//[18] ST1 SWORD
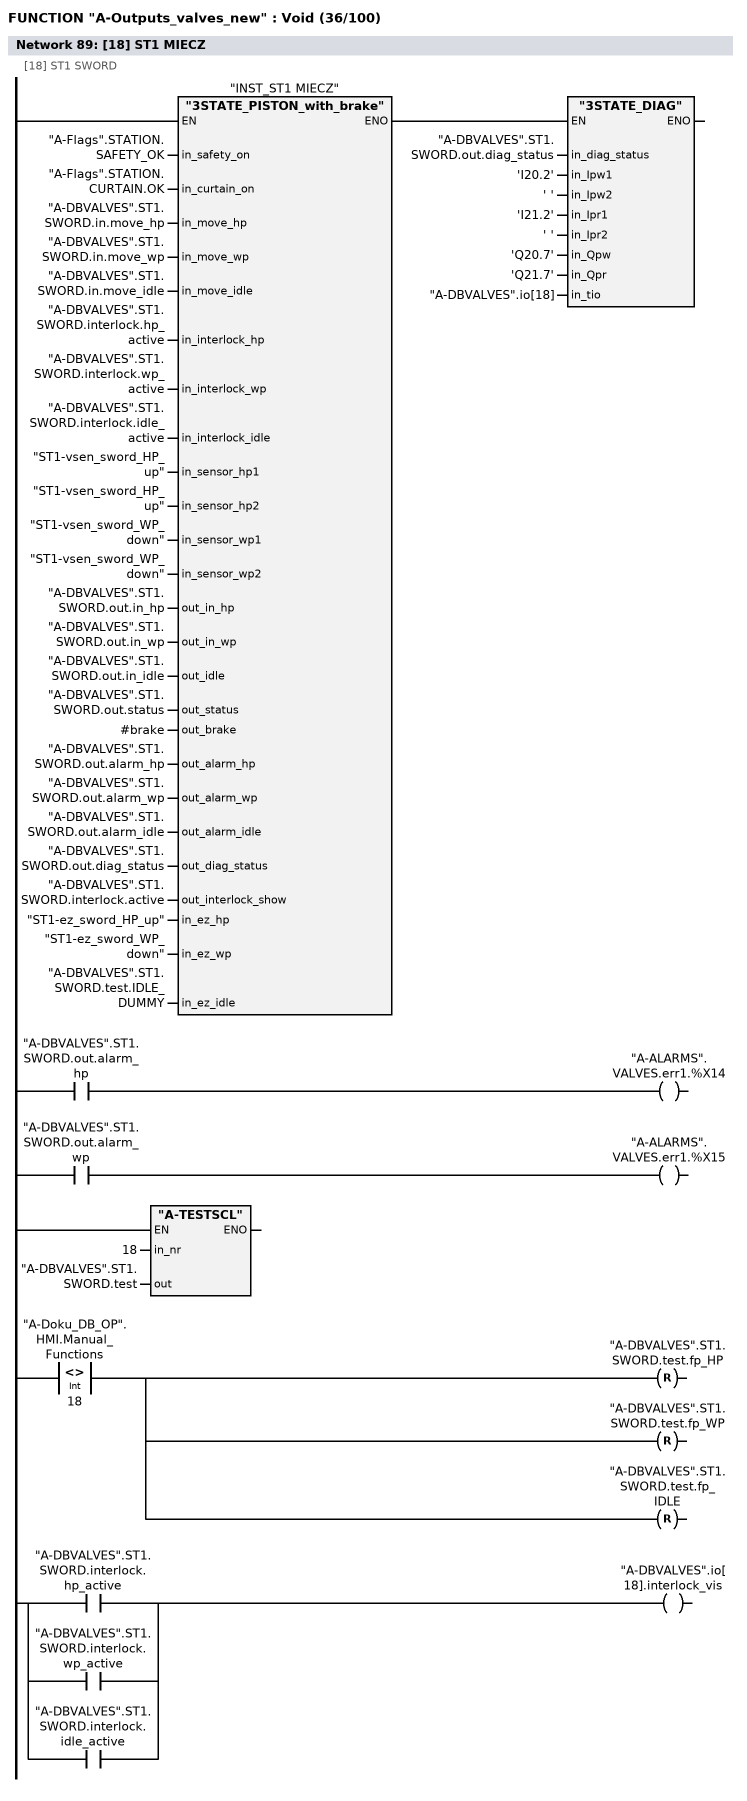
      CALL "3STATE_PISTON_with_brake", "INST_ST1 MIECZ"
      (  in_safety_on                := "A-Flags".STATION.SAFETY_OK ,
         in_curtain_on               := "A-Flags".STATION.CURTAIN.OK ,
         in_move_hp                  := "A-DBVALVES".ST1.SWORD.in.move_hp ,
         in_move_wp                  := "A-DBVALVES".ST1.SWORD.in.move_wp ,
         in_move_idle                := "A-DBVALVES".ST1.SWORD.in.move_idle ,
         in_interlock_hp             := "A-DBVALVES".ST1.SWORD.interlock.hp_active ,
         in_interlock_wp             := "A-DBVALVES".ST1.SWORD.interlock.wp_active ,
         in_interlock_idle           := "A-DBVALVES".ST1.SWORD.interlock.idle_active ,
         in_sensor_hp1               := "ST1-vsen_sword_HP_up" ,
         in_sensor_hp2               := "ST1-vsen_sword_HP_up" ,
         in_sensor_wp1               := "ST1-vsen_sword_WP_down" ,
         in_sensor_wp2               := "ST1-vsen_sword_WP_down" ,
         out_in_hp                   := "A-DBVALVES".ST1.SWORD.out.in_hp ,
         out_in_wp                   := "A-DBVALVES".ST1.SWORD.out.in_wp ,
         out_idle                    := "A-DBVALVES".ST1.SWORD.out.in_idle ,
         out_status                  := "A-DBVALVES".ST1.SWORD.out.status ,
         out_brake                   := #brake ,
         out_alarm_hp                := "A-DBVALVES".ST1.SWORD.out.alarm_hp ,
         out_alarm_wp                := "A-DBVALVES".ST1.SWORD.out.alarm_wp ,
         out_alarm_idle              := "A-DBVALVES".ST1.SWORD.out.alarm_idle ,
         out_diag_status             := "A-DBVALVES".ST1.SWORD.out.diag_status ,
         out_interlock_show          := "A-DBVALVES".ST1.SWORD.interlock.active ,
         in_ez_hp                    := "ST1-ez_sword_HP_up" ,
         in_ez_wp                    := "ST1-ez_sword_WP_down" ,
         in_ez_idle                  := "A-DBVALVES".ST1.SWORD.test.IDLE_DUMMY
      );

      CALL "3STATE_DIAG"
      (  in_diag_status              := "A-DBVALVES".ST1.SWORD.out.diag_status ,
         in_Ipw1                     := 'I20.2' ,
         in_Ipw2                     := ' ' ,
         in_Ipr1                     := 'I21.2' ,
         in_Ipr2                     := ' ' ,
         in_Qpw                      := 'Q20.7' ,
         in_Qpr                      := 'Q21.7' ,
         in_tio                      := "A-DBVALVES".io[18]
      );

      A "A-DBVALVES".ST1.SWORD.out.alarm_hp;
      = "A-ALARMS".VALVES.err1.%X14;

      A "A-DBVALVES".ST1.SWORD.out.alarm_wp;
      = "A-ALARMS".VALVES.err1.%X15;

      CALL "A-TESTSCL"
      (  in_nr                       := 18 ,
         out                         := "A-DBVALVES".ST1.SWORD.test
      );

      A(;
      L "A-Doku_DB_OP".HMI.Manual_Functions;
      L 18;
      <>I;
      );
      R "A-DBVALVES".ST1.SWORD.test.fp_HP;
      R "A-DBVALVES".ST1.SWORD.test.fp_WP;
      R "A-DBVALVES".ST1.SWORD.test.fp_IDLE;

      O "A-DBVALVES".ST1.SWORD.interlock.hp_active;
      O "A-DBVALVES".ST1.SWORD.interlock.wp_active;
      O "A-DBVALVES".ST1.SWORD.interlock.idle_active;
      = "A-DBVALVES".io[18].interlock_vis;
NETWORK
TITLE = -

NETWORK
TITLE = [19] ST2 STACJA_PRZESUW - HP
//[19] ST2 STATION_MOVEMENT - HP
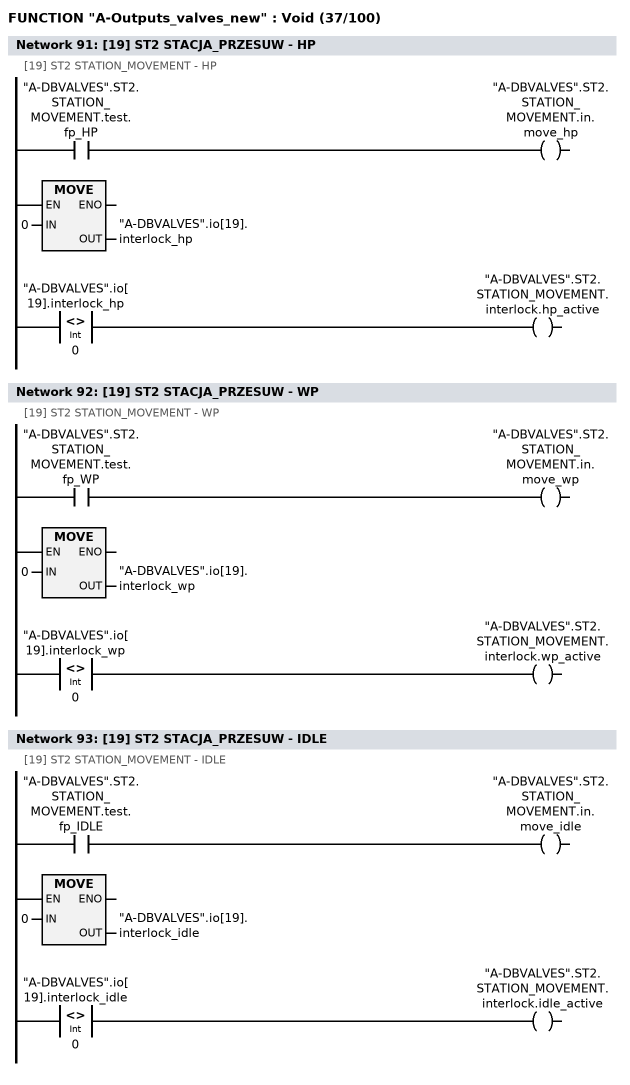
      O "A-DBVALVES".ST2.STATION_MOVEMENT.test.fp_HP;
//    O     "A-Flags".STATION.IN_HP_STEP
      = "A-DBVALVES".ST2.STATION_MOVEMENT.in.move_hp;

// Interlock hp
      L 0;
      T "A-DBVALVES".io[19].interlock_hp;

//{INTERLOCK_HP19}

      A(;
      L "A-DBVALVES".io[19].interlock_hp;
      L 0;
      <>I;
      );
      = "A-DBVALVES".ST2.STATION_MOVEMENT.interlock.hp_active;
NETWORK
TITLE = [19] ST2 STACJA_PRZESUW - WP
//[19] ST2 STATION_MOVEMENT - WP
      O "A-DBVALVES".ST2.STATION_MOVEMENT.test.fp_WP;
      = "A-DBVALVES".ST2.STATION_MOVEMENT.in.move_wp;

// Interlock wp
      L 0;
      T "A-DBVALVES".io[19].interlock_wp;

//{INTERLOCK_WP19}

      A(;
      L "A-DBVALVES".io[19].interlock_wp;
      L 0;
      <>I;
      );
      = "A-DBVALVES".ST2.STATION_MOVEMENT.interlock.wp_active;
NETWORK
TITLE = [19] ST2 STACJA_PRZESUW - IDLE
//[19] ST2 STATION_MOVEMENT - IDLE
      O "A-DBVALVES".ST2.STATION_MOVEMENT.test.fp_IDLE;
      = "A-DBVALVES".ST2.STATION_MOVEMENT.in.move_idle;

// Interlock idle
      L 0;
      T "A-DBVALVES".io[19].interlock_idle;

//{INTERLOCK_IDLE19}

      A(;
      L "A-DBVALVES".io[19].interlock_idle;
      L 0;
      <>I;
      );
      = "A-DBVALVES".ST2.STATION_MOVEMENT.interlock.idle_active;
NETWORK
TITLE = [19] ST2 STACJA_PRZESUW
//[19] ST2 STATION_MOVEMENT
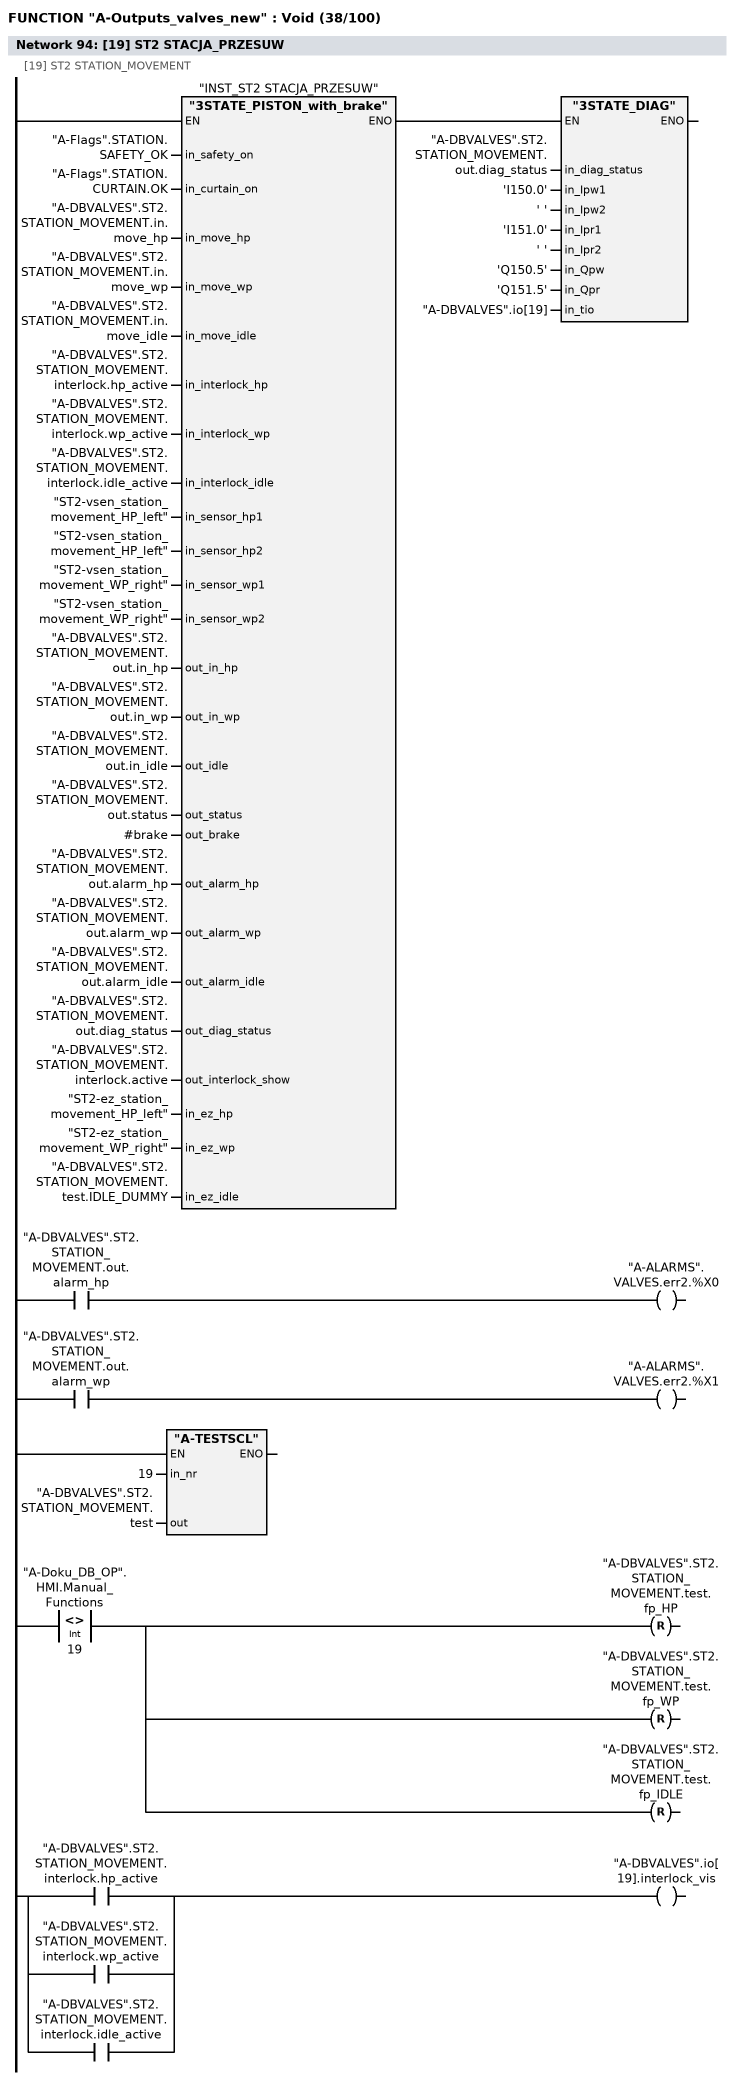
      CALL "3STATE_PISTON_with_brake", "INST_ST2 STACJA_PRZESUW"
      (  in_safety_on                := "A-Flags".STATION.SAFETY_OK ,
         in_curtain_on               := "A-Flags".STATION.CURTAIN.OK ,
         in_move_hp                  := "A-DBVALVES".ST2.STATION_MOVEMENT.in.move_hp ,
         in_move_wp                  := "A-DBVALVES".ST2.STATION_MOVEMENT.in.move_wp ,
         in_move_idle                := "A-DBVALVES".ST2.STATION_MOVEMENT.in.move_idle ,
         in_interlock_hp             := "A-DBVALVES".ST2.STATION_MOVEMENT.interlock.hp_active ,
         in_interlock_wp             := "A-DBVALVES".ST2.STATION_MOVEMENT.interlock.wp_active ,
         in_interlock_idle           := "A-DBVALVES".ST2.STATION_MOVEMENT.interlock.idle_active ,
         in_sensor_hp1               := "ST2-vsen_station_movement_HP_left" ,
         in_sensor_hp2               := "ST2-vsen_station_movement_HP_left" ,
         in_sensor_wp1               := "ST2-vsen_station_movement_WP_right" ,
         in_sensor_wp2               := "ST2-vsen_station_movement_WP_right" ,
         out_in_hp                   := "A-DBVALVES".ST2.STATION_MOVEMENT.out.in_hp ,
         out_in_wp                   := "A-DBVALVES".ST2.STATION_MOVEMENT.out.in_wp ,
         out_idle                    := "A-DBVALVES".ST2.STATION_MOVEMENT.out.in_idle ,
         out_status                  := "A-DBVALVES".ST2.STATION_MOVEMENT.out.status ,
         out_brake                   := #brake ,
         out_alarm_hp                := "A-DBVALVES".ST2.STATION_MOVEMENT.out.alarm_hp ,
         out_alarm_wp                := "A-DBVALVES".ST2.STATION_MOVEMENT.out.alarm_wp ,
         out_alarm_idle              := "A-DBVALVES".ST2.STATION_MOVEMENT.out.alarm_idle ,
         out_diag_status             := "A-DBVALVES".ST2.STATION_MOVEMENT.out.diag_status ,
         out_interlock_show          := "A-DBVALVES".ST2.STATION_MOVEMENT.interlock.active ,
         in_ez_hp                    := "ST2-ez_station_movement_HP_left" ,
         in_ez_wp                    := "ST2-ez_station_movement_WP_right" ,
         in_ez_idle                  := "A-DBVALVES".ST2.STATION_MOVEMENT.test.IDLE_DUMMY
      );

      CALL "3STATE_DIAG"
      (  in_diag_status              := "A-DBVALVES".ST2.STATION_MOVEMENT.out.diag_status ,
         in_Ipw1                     := 'I150.0' ,
         in_Ipw2                     := ' ' ,
         in_Ipr1                     := 'I151.0' ,
         in_Ipr2                     := ' ' ,
         in_Qpw                      := 'Q150.5' ,
         in_Qpr                      := 'Q151.5' ,
         in_tio                      := "A-DBVALVES".io[19]
      );

      A "A-DBVALVES".ST2.STATION_MOVEMENT.out.alarm_hp;
      = "A-ALARMS".VALVES.err2.%X0;

      A "A-DBVALVES".ST2.STATION_MOVEMENT.out.alarm_wp;
      = "A-ALARMS".VALVES.err2.%X1;

      CALL "A-TESTSCL"
      (  in_nr                       := 19 ,
         out                         := "A-DBVALVES".ST2.STATION_MOVEMENT.test
      );

      A(;
      L "A-Doku_DB_OP".HMI.Manual_Functions;
      L 19;
      <>I;
      );
      R "A-DBVALVES".ST2.STATION_MOVEMENT.test.fp_HP;
      R "A-DBVALVES".ST2.STATION_MOVEMENT.test.fp_WP;
      R "A-DBVALVES".ST2.STATION_MOVEMENT.test.fp_IDLE;

      O "A-DBVALVES".ST2.STATION_MOVEMENT.interlock.hp_active;
      O "A-DBVALVES".ST2.STATION_MOVEMENT.interlock.wp_active;
      O "A-DBVALVES".ST2.STATION_MOVEMENT.interlock.idle_active;
      = "A-DBVALVES".io[19].interlock_vis;
NETWORK
TITLE = -

NETWORK
TITLE = [20] ST2 MIECZ_WYSUW - HP
//[20] ST2 SWORD_SLIDE_OUT - HP
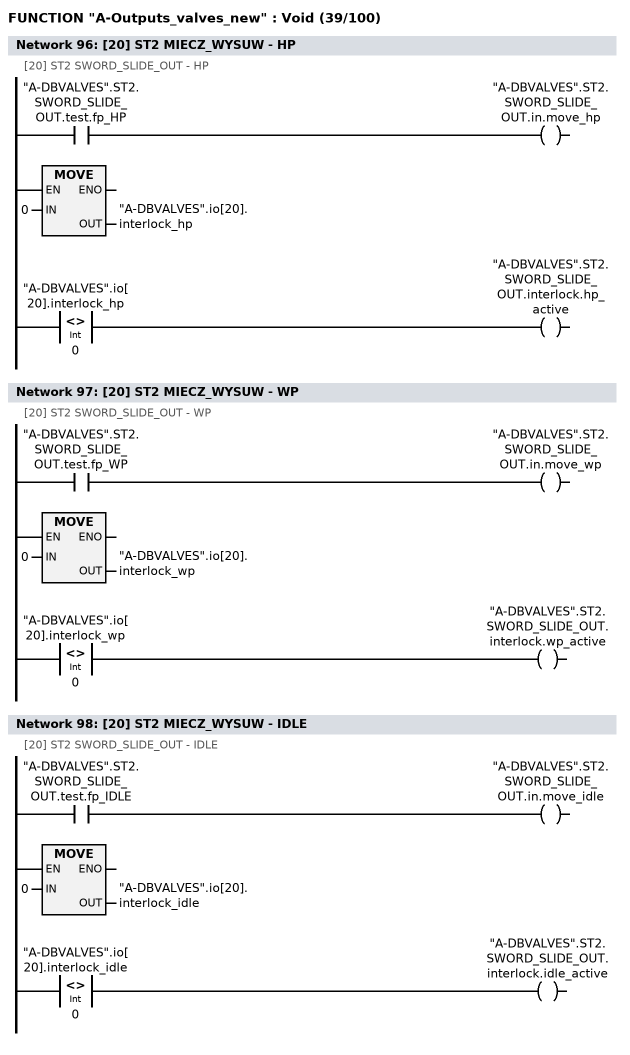
      O "A-DBVALVES".ST2.SWORD_SLIDE_OUT.test.fp_HP;
//    O     "A-Flags".STATION.IN_HP_STEP
      = "A-DBVALVES".ST2.SWORD_SLIDE_OUT.in.move_hp;

// Interlock hp
      L 0;
      T "A-DBVALVES".io[20].interlock_hp;

//{INTERLOCK_HP20}

      A(;
      L "A-DBVALVES".io[20].interlock_hp;
      L 0;
      <>I;
      );
      = "A-DBVALVES".ST2.SWORD_SLIDE_OUT.interlock.hp_active;
NETWORK
TITLE = [20] ST2 MIECZ_WYSUW - WP
//[20] ST2 SWORD_SLIDE_OUT - WP
      O "A-DBVALVES".ST2.SWORD_SLIDE_OUT.test.fp_WP;
      = "A-DBVALVES".ST2.SWORD_SLIDE_OUT.in.move_wp;

// Interlock wp
      L 0;
      T "A-DBVALVES".io[20].interlock_wp;

//{INTERLOCK_WP20}

      A(;
      L "A-DBVALVES".io[20].interlock_wp;
      L 0;
      <>I;
      );
      = "A-DBVALVES".ST2.SWORD_SLIDE_OUT.interlock.wp_active;
NETWORK
TITLE = [20] ST2 MIECZ_WYSUW - IDLE
//[20] ST2 SWORD_SLIDE_OUT - IDLE
      O "A-DBVALVES".ST2.SWORD_SLIDE_OUT.test.fp_IDLE;
      = "A-DBVALVES".ST2.SWORD_SLIDE_OUT.in.move_idle;

// Interlock idle
      L 0;
      T "A-DBVALVES".io[20].interlock_idle;

//{INTERLOCK_IDLE20}

      A(;
      L "A-DBVALVES".io[20].interlock_idle;
      L 0;
      <>I;
      );
      = "A-DBVALVES".ST2.SWORD_SLIDE_OUT.interlock.idle_active;
NETWORK
TITLE = [20] ST2 MIECZ_WYSUW
//[20] ST2 SWORD_SLIDE_OUT
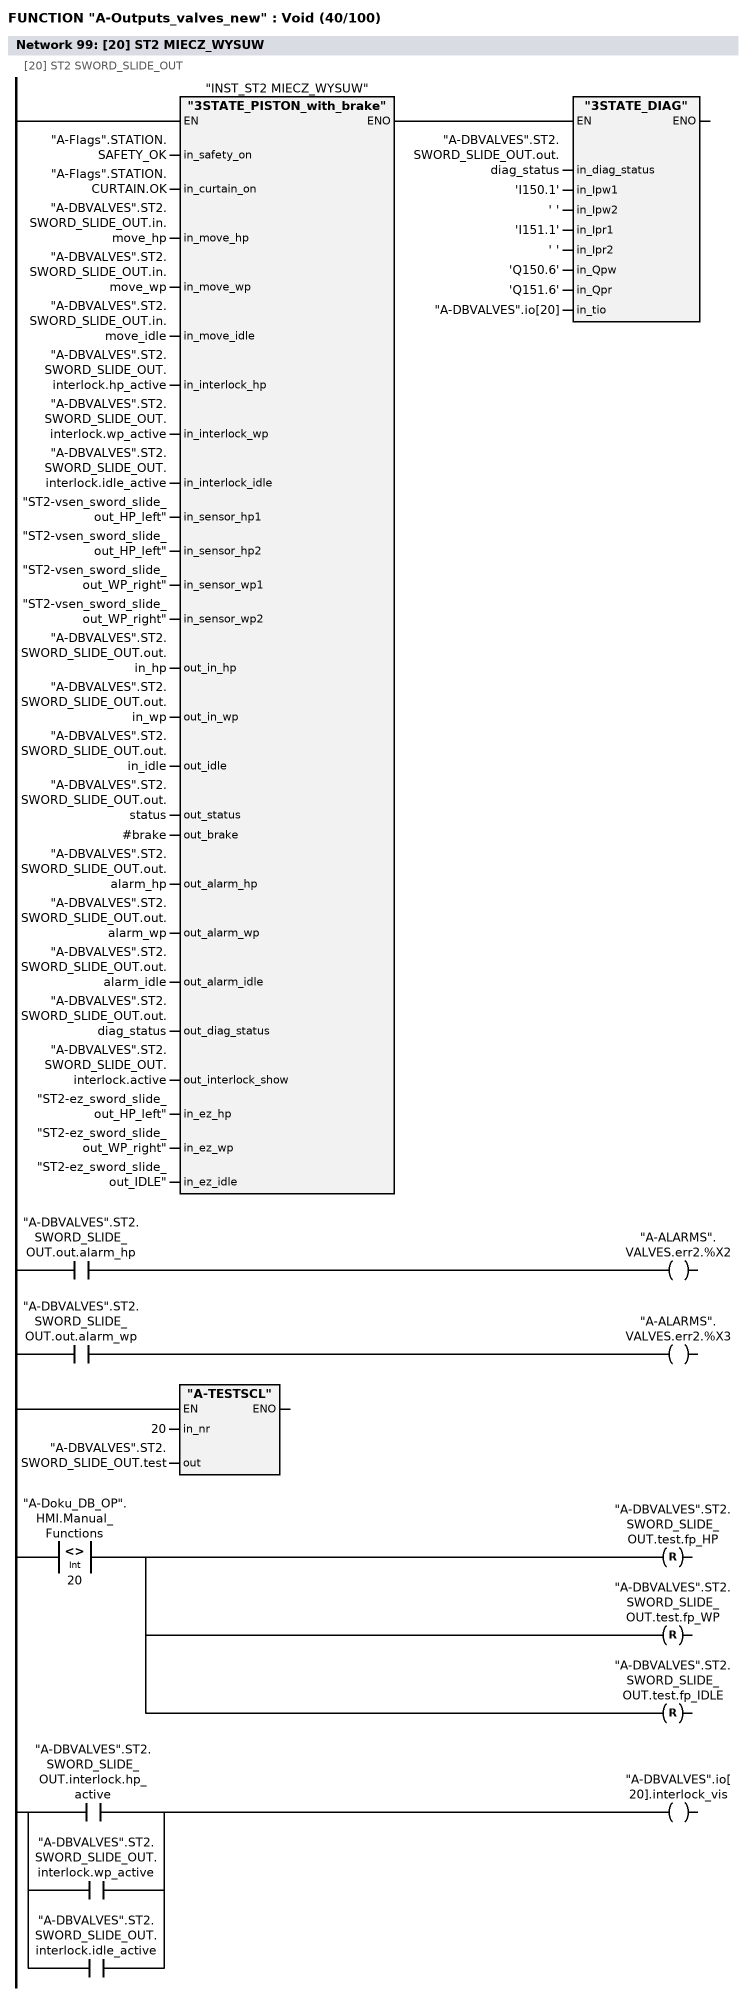
      CALL "3STATE_PISTON_with_brake", "INST_ST2 MIECZ_WYSUW"
      (  in_safety_on                := "A-Flags".STATION.SAFETY_OK ,
         in_curtain_on               := "A-Flags".STATION.CURTAIN.OK ,
         in_move_hp                  := "A-DBVALVES".ST2.SWORD_SLIDE_OUT.in.move_hp ,
         in_move_wp                  := "A-DBVALVES".ST2.SWORD_SLIDE_OUT.in.move_wp ,
         in_move_idle                := "A-DBVALVES".ST2.SWORD_SLIDE_OUT.in.move_idle ,
         in_interlock_hp             := "A-DBVALVES".ST2.SWORD_SLIDE_OUT.interlock.hp_active ,
         in_interlock_wp             := "A-DBVALVES".ST2.SWORD_SLIDE_OUT.interlock.wp_active ,
         in_interlock_idle           := "A-DBVALVES".ST2.SWORD_SLIDE_OUT.interlock.idle_active ,
         in_sensor_hp1               := "ST2-vsen_sword_slide_out_HP_left" ,
         in_sensor_hp2               := "ST2-vsen_sword_slide_out_HP_left" ,
         in_sensor_wp1               := "ST2-vsen_sword_slide_out_WP_right" ,
         in_sensor_wp2               := "ST2-vsen_sword_slide_out_WP_right" ,
         out_in_hp                   := "A-DBVALVES".ST2.SWORD_SLIDE_OUT.out.in_hp ,
         out_in_wp                   := "A-DBVALVES".ST2.SWORD_SLIDE_OUT.out.in_wp ,
         out_idle                    := "A-DBVALVES".ST2.SWORD_SLIDE_OUT.out.in_idle ,
         out_status                  := "A-DBVALVES".ST2.SWORD_SLIDE_OUT.out.status ,
         out_brake                   := #brake ,
         out_alarm_hp                := "A-DBVALVES".ST2.SWORD_SLIDE_OUT.out.alarm_hp ,
         out_alarm_wp                := "A-DBVALVES".ST2.SWORD_SLIDE_OUT.out.alarm_wp ,
         out_alarm_idle              := "A-DBVALVES".ST2.SWORD_SLIDE_OUT.out.alarm_idle ,
         out_diag_status             := "A-DBVALVES".ST2.SWORD_SLIDE_OUT.out.diag_status ,
         out_interlock_show          := "A-DBVALVES".ST2.SWORD_SLIDE_OUT.interlock.active ,
         in_ez_hp                    := "ST2-ez_sword_slide_out_HP_left" ,
         in_ez_wp                    := "ST2-ez_sword_slide_out_WP_right" ,
         in_ez_idle                  := "ST2-ez_sword_slide_out_IDLE"
      );

      CALL "3STATE_DIAG"
      (  in_diag_status              := "A-DBVALVES".ST2.SWORD_SLIDE_OUT.out.diag_status ,
         in_Ipw1                     := 'I150.1' ,
         in_Ipw2                     := ' ' ,
         in_Ipr1                     := 'I151.1' ,
         in_Ipr2                     := ' ' ,
         in_Qpw                      := 'Q150.6' ,
         in_Qpr                      := 'Q151.6' ,
         in_tio                      := "A-DBVALVES".io[20]
      );

      A "A-DBVALVES".ST2.SWORD_SLIDE_OUT.out.alarm_hp;
      = "A-ALARMS".VALVES.err2.%X2;

      A "A-DBVALVES".ST2.SWORD_SLIDE_OUT.out.alarm_wp;
      = "A-ALARMS".VALVES.err2.%X3;

      CALL "A-TESTSCL"
      (  in_nr                       := 20 ,
         out                         := "A-DBVALVES".ST2.SWORD_SLIDE_OUT.test
      );

      A(;
      L "A-Doku_DB_OP".HMI.Manual_Functions;
      L 20;
      <>I;
      );
      R "A-DBVALVES".ST2.SWORD_SLIDE_OUT.test.fp_HP;
      R "A-DBVALVES".ST2.SWORD_SLIDE_OUT.test.fp_WP;
      R "A-DBVALVES".ST2.SWORD_SLIDE_OUT.test.fp_IDLE;

      O "A-DBVALVES".ST2.SWORD_SLIDE_OUT.interlock.hp_active;
      O "A-DBVALVES".ST2.SWORD_SLIDE_OUT.interlock.wp_active;
      O "A-DBVALVES".ST2.SWORD_SLIDE_OUT.interlock.idle_active;
      = "A-DBVALVES".io[20].interlock_vis;
NETWORK
TITLE = -

NETWORK
TITLE = [21] ST2 MIECZ - HP
//[21] ST2 SWORD - HP
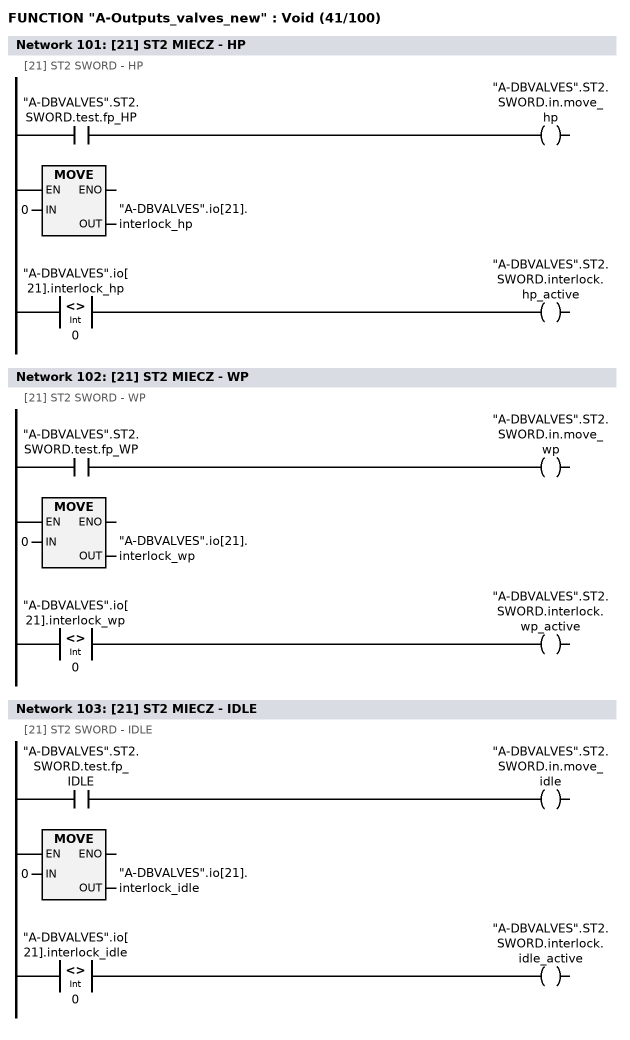
      O "A-DBVALVES".ST2.SWORD.test.fp_HP;
//    O     "A-Flags".STATION.IN_HP_STEP
      = "A-DBVALVES".ST2.SWORD.in.move_hp;

// Interlock hp
      L 0;
      T "A-DBVALVES".io[21].interlock_hp;

//{INTERLOCK_HP21}

      A(;
      L "A-DBVALVES".io[21].interlock_hp;
      L 0;
      <>I;
      );
      = "A-DBVALVES".ST2.SWORD.interlock.hp_active;
NETWORK
TITLE = [21] ST2 MIECZ - WP
//[21] ST2 SWORD - WP
      O "A-DBVALVES".ST2.SWORD.test.fp_WP;
      = "A-DBVALVES".ST2.SWORD.in.move_wp;

// Interlock wp
      L 0;
      T "A-DBVALVES".io[21].interlock_wp;

//{INTERLOCK_WP21}

      A(;
      L "A-DBVALVES".io[21].interlock_wp;
      L 0;
      <>I;
      );
      = "A-DBVALVES".ST2.SWORD.interlock.wp_active;
NETWORK
TITLE = [21] ST2 MIECZ - IDLE
//[21] ST2 SWORD - IDLE
      O "A-DBVALVES".ST2.SWORD.test.fp_IDLE;
      = "A-DBVALVES".ST2.SWORD.in.move_idle;

// Interlock idle
      L 0;
      T "A-DBVALVES".io[21].interlock_idle;

//{INTERLOCK_IDLE21}

      A(;
      L "A-DBVALVES".io[21].interlock_idle;
      L 0;
      <>I;
      );
      = "A-DBVALVES".ST2.SWORD.interlock.idle_active;
NETWORK
TITLE = [21] ST2 MIECZ
//[21] ST2 SWORD
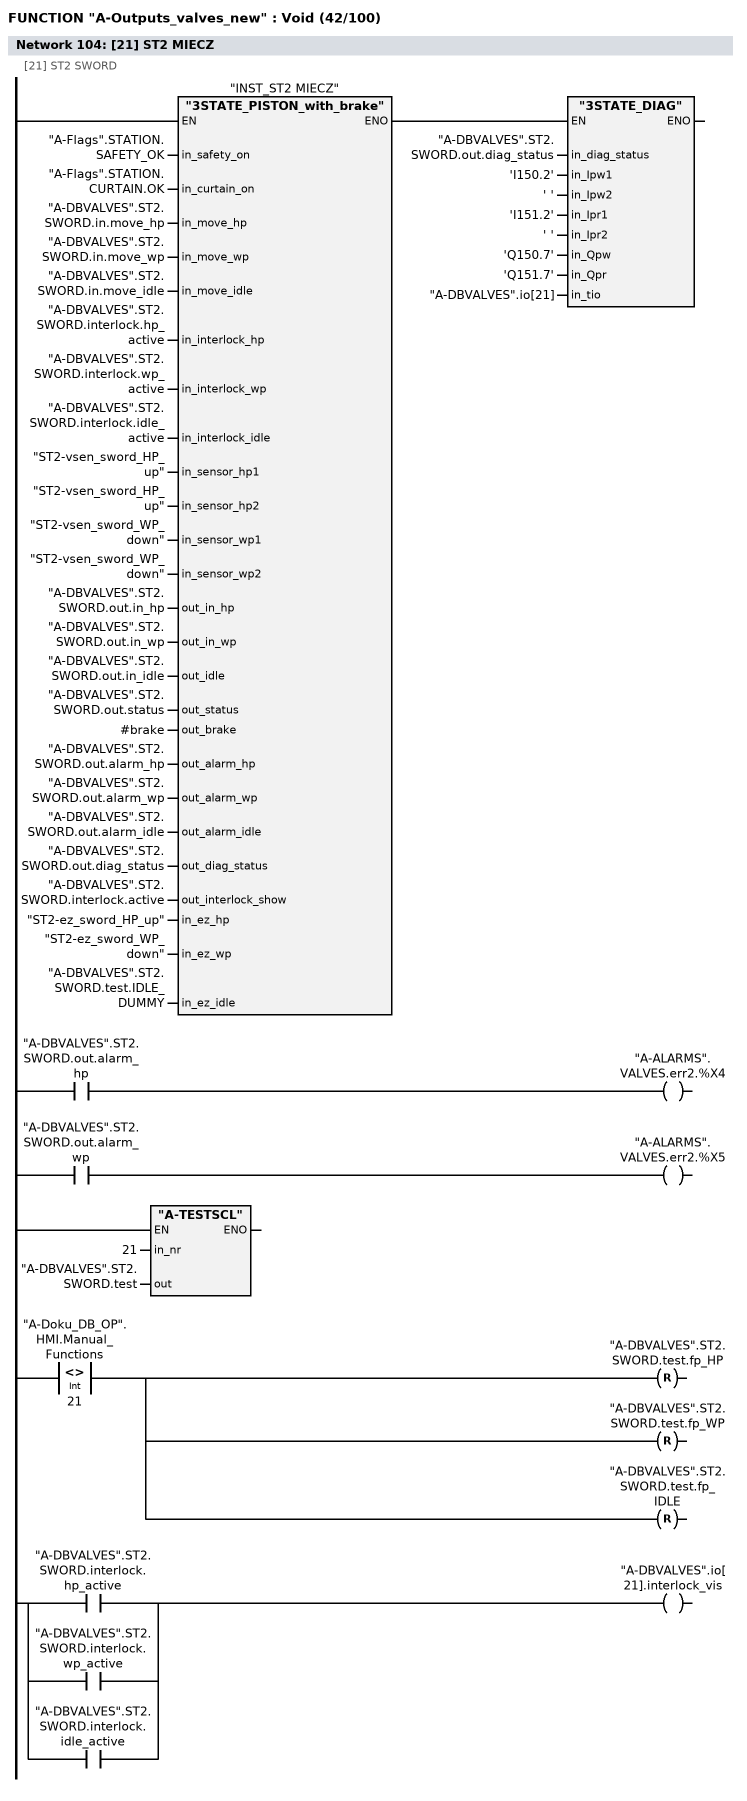
      CALL "3STATE_PISTON_with_brake", "INST_ST2 MIECZ"
      (  in_safety_on                := "A-Flags".STATION.SAFETY_OK ,
         in_curtain_on               := "A-Flags".STATION.CURTAIN.OK ,
         in_move_hp                  := "A-DBVALVES".ST2.SWORD.in.move_hp ,
         in_move_wp                  := "A-DBVALVES".ST2.SWORD.in.move_wp ,
         in_move_idle                := "A-DBVALVES".ST2.SWORD.in.move_idle ,
         in_interlock_hp             := "A-DBVALVES".ST2.SWORD.interlock.hp_active ,
         in_interlock_wp             := "A-DBVALVES".ST2.SWORD.interlock.wp_active ,
         in_interlock_idle           := "A-DBVALVES".ST2.SWORD.interlock.idle_active ,
         in_sensor_hp1               := "ST2-vsen_sword_HP_up" ,
         in_sensor_hp2               := "ST2-vsen_sword_HP_up" ,
         in_sensor_wp1               := "ST2-vsen_sword_WP_down" ,
         in_sensor_wp2               := "ST2-vsen_sword_WP_down" ,
         out_in_hp                   := "A-DBVALVES".ST2.SWORD.out.in_hp ,
         out_in_wp                   := "A-DBVALVES".ST2.SWORD.out.in_wp ,
         out_idle                    := "A-DBVALVES".ST2.SWORD.out.in_idle ,
         out_status                  := "A-DBVALVES".ST2.SWORD.out.status ,
         out_brake                   := #brake ,
         out_alarm_hp                := "A-DBVALVES".ST2.SWORD.out.alarm_hp ,
         out_alarm_wp                := "A-DBVALVES".ST2.SWORD.out.alarm_wp ,
         out_alarm_idle              := "A-DBVALVES".ST2.SWORD.out.alarm_idle ,
         out_diag_status             := "A-DBVALVES".ST2.SWORD.out.diag_status ,
         out_interlock_show          := "A-DBVALVES".ST2.SWORD.interlock.active ,
         in_ez_hp                    := "ST2-ez_sword_HP_up" ,
         in_ez_wp                    := "ST2-ez_sword_WP_down" ,
         in_ez_idle                  := "A-DBVALVES".ST2.SWORD.test.IDLE_DUMMY
      );

      CALL "3STATE_DIAG"
      (  in_diag_status              := "A-DBVALVES".ST2.SWORD.out.diag_status ,
         in_Ipw1                     := 'I150.2' ,
         in_Ipw2                     := ' ' ,
         in_Ipr1                     := 'I151.2' ,
         in_Ipr2                     := ' ' ,
         in_Qpw                      := 'Q150.7' ,
         in_Qpr                      := 'Q151.7' ,
         in_tio                      := "A-DBVALVES".io[21]
      );

      A "A-DBVALVES".ST2.SWORD.out.alarm_hp;
      = "A-ALARMS".VALVES.err2.%X4;

      A "A-DBVALVES".ST2.SWORD.out.alarm_wp;
      = "A-ALARMS".VALVES.err2.%X5;

      CALL "A-TESTSCL"
      (  in_nr                       := 21 ,
         out                         := "A-DBVALVES".ST2.SWORD.test
      );

      A(;
      L "A-Doku_DB_OP".HMI.Manual_Functions;
      L 21;
      <>I;
      );
      R "A-DBVALVES".ST2.SWORD.test.fp_HP;
      R "A-DBVALVES".ST2.SWORD.test.fp_WP;
      R "A-DBVALVES".ST2.SWORD.test.fp_IDLE;

      O "A-DBVALVES".ST2.SWORD.interlock.hp_active;
      O "A-DBVALVES".ST2.SWORD.interlock.wp_active;
      O "A-DBVALVES".ST2.SWORD.interlock.idle_active;
      = "A-DBVALVES".io[21].interlock_vis;
NETWORK
TITLE = -

NETWORK
TITLE = [22] ST3 MIECZ_PODNOSZENIE - HP
//[22] ST3 SWORD_RISING - HP
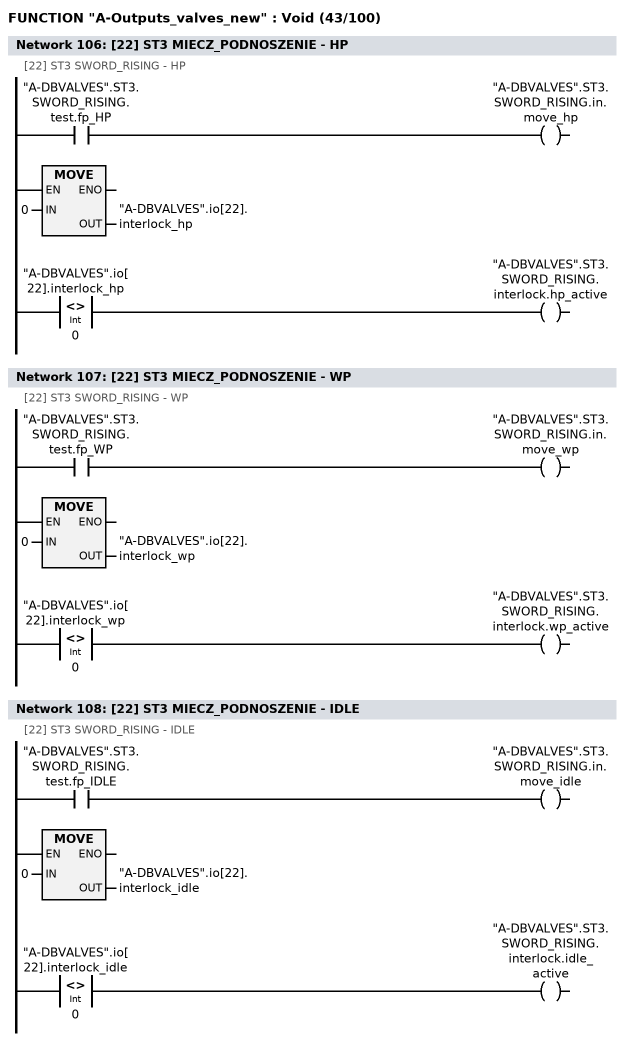
      O "A-DBVALVES".ST3.SWORD_RISING.test.fp_HP;
//    O     "A-Flags".STATION.IN_HP_STEP
      = "A-DBVALVES".ST3.SWORD_RISING.in.move_hp;

// Interlock hp
      L 0;
      T "A-DBVALVES".io[22].interlock_hp;

//{INTERLOCK_HP22}

      A(;
      L "A-DBVALVES".io[22].interlock_hp;
      L 0;
      <>I;
      );
      = "A-DBVALVES".ST3.SWORD_RISING.interlock.hp_active;
NETWORK
TITLE = [22] ST3 MIECZ_PODNOSZENIE - WP
//[22] ST3 SWORD_RISING - WP
      O "A-DBVALVES".ST3.SWORD_RISING.test.fp_WP;
      = "A-DBVALVES".ST3.SWORD_RISING.in.move_wp;

// Interlock wp
      L 0;
      T "A-DBVALVES".io[22].interlock_wp;

//{INTERLOCK_WP22}

      A(;
      L "A-DBVALVES".io[22].interlock_wp;
      L 0;
      <>I;
      );
      = "A-DBVALVES".ST3.SWORD_RISING.interlock.wp_active;
NETWORK
TITLE = [22] ST3 MIECZ_PODNOSZENIE - IDLE
//[22] ST3 SWORD_RISING - IDLE
      O "A-DBVALVES".ST3.SWORD_RISING.test.fp_IDLE;
      = "A-DBVALVES".ST3.SWORD_RISING.in.move_idle;

// Interlock idle
      L 0;
      T "A-DBVALVES".io[22].interlock_idle;

//{INTERLOCK_IDLE22}

      A(;
      L "A-DBVALVES".io[22].interlock_idle;
      L 0;
      <>I;
      );
      = "A-DBVALVES".ST3.SWORD_RISING.interlock.idle_active;
NETWORK
TITLE = [22] ST3 MIECZ_PODNOSZENIE
//[22] ST3 SWORD_RISING
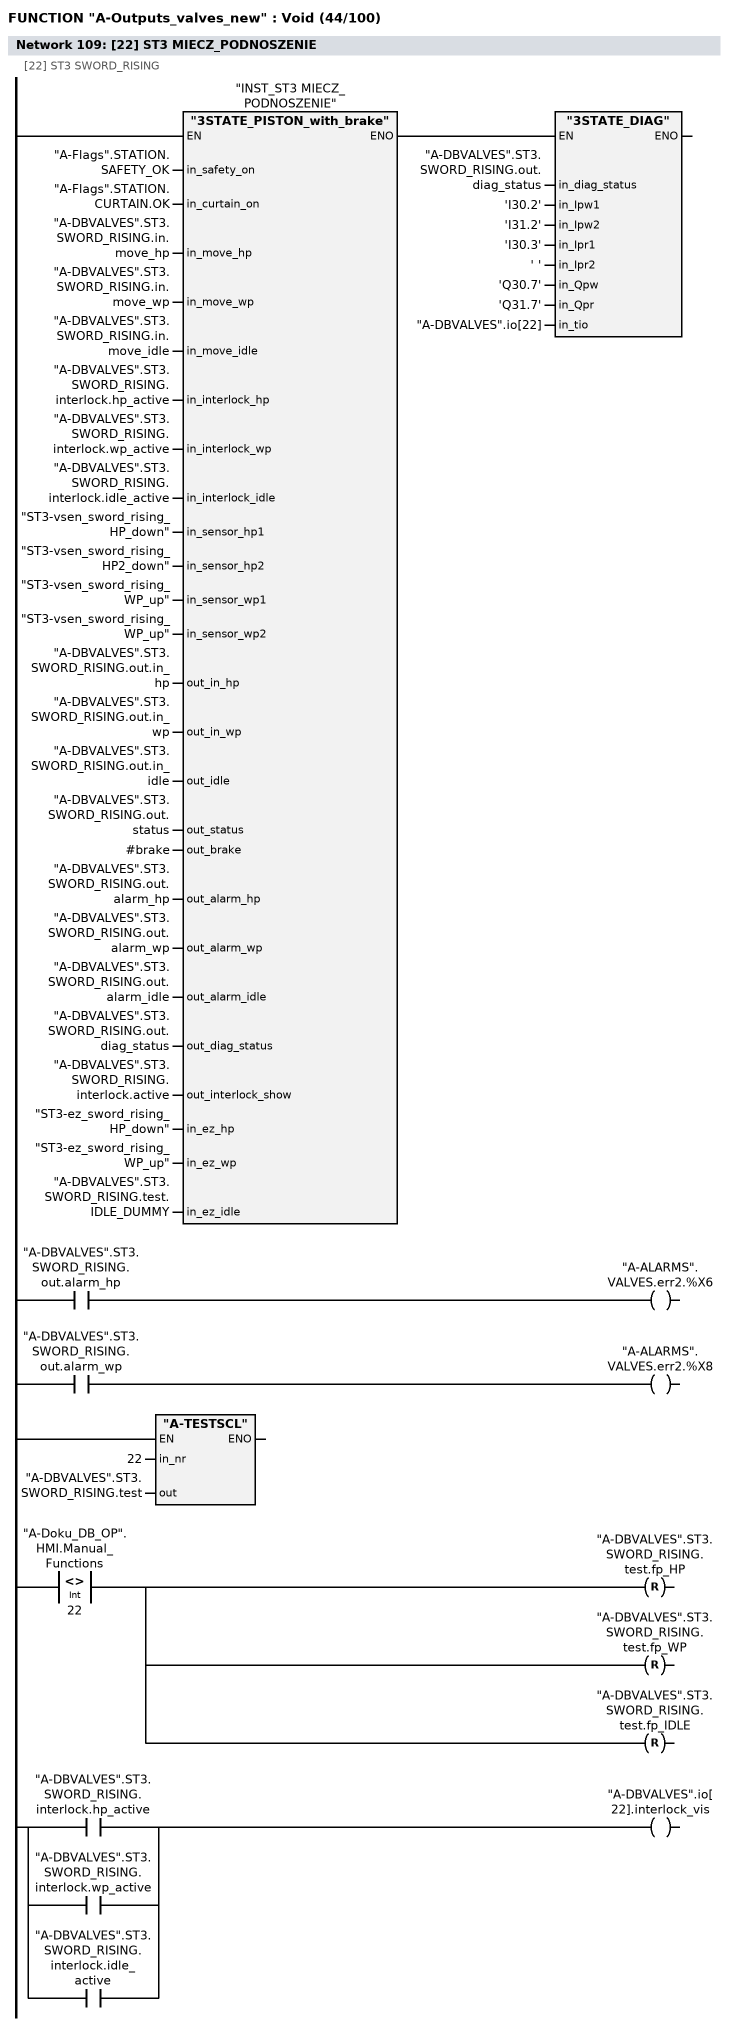
      CALL "3STATE_PISTON_with_brake", "INST_ST3 MIECZ_PODNOSZENIE"
      (  in_safety_on                := "A-Flags".STATION.SAFETY_OK ,
         in_curtain_on               := "A-Flags".STATION.CURTAIN.OK ,
         in_move_hp                  := "A-DBVALVES".ST3.SWORD_RISING.in.move_hp ,
         in_move_wp                  := "A-DBVALVES".ST3.SWORD_RISING.in.move_wp ,
         in_move_idle                := "A-DBVALVES".ST3.SWORD_RISING.in.move_idle ,
         in_interlock_hp             := "A-DBVALVES".ST3.SWORD_RISING.interlock.hp_active ,
         in_interlock_wp             := "A-DBVALVES".ST3.SWORD_RISING.interlock.wp_active ,
         in_interlock_idle           := "A-DBVALVES".ST3.SWORD_RISING.interlock.idle_active ,
         in_sensor_hp1               := "ST3-vsen_sword_rising_HP_down" ,
         in_sensor_hp2               := "ST3-vsen_sword_rising_HP2_down" ,
         in_sensor_wp1               := "ST3-vsen_sword_rising_WP_up" ,
         in_sensor_wp2               := "ST3-vsen_sword_rising_WP_up" ,
         out_in_hp                   := "A-DBVALVES".ST3.SWORD_RISING.out.in_hp ,
         out_in_wp                   := "A-DBVALVES".ST3.SWORD_RISING.out.in_wp ,
         out_idle                    := "A-DBVALVES".ST3.SWORD_RISING.out.in_idle ,
         out_status                  := "A-DBVALVES".ST3.SWORD_RISING.out.status ,
         out_brake                   := #brake ,
         out_alarm_hp                := "A-DBVALVES".ST3.SWORD_RISING.out.alarm_hp ,
         out_alarm_wp                := "A-DBVALVES".ST3.SWORD_RISING.out.alarm_wp ,
         out_alarm_idle              := "A-DBVALVES".ST3.SWORD_RISING.out.alarm_idle ,
         out_diag_status             := "A-DBVALVES".ST3.SWORD_RISING.out.diag_status ,
         out_interlock_show          := "A-DBVALVES".ST3.SWORD_RISING.interlock.active ,
         in_ez_hp                    := "ST3-ez_sword_rising_HP_down" ,
         in_ez_wp                    := "ST3-ez_sword_rising_WP_up" ,
         in_ez_idle                  := "A-DBVALVES".ST3.SWORD_RISING.test.IDLE_DUMMY
      );

      CALL "3STATE_DIAG"
      (  in_diag_status              := "A-DBVALVES".ST3.SWORD_RISING.out.diag_status ,
         in_Ipw1                     := 'I30.2' ,
         in_Ipw2                     := 'I31.2' ,
         in_Ipr1                     := 'I30.3' ,
         in_Ipr2                     := ' ' ,
         in_Qpw                      := 'Q30.7' ,
         in_Qpr                      := 'Q31.7' ,
         in_tio                      := "A-DBVALVES".io[22]
      );

      A "A-DBVALVES".ST3.SWORD_RISING.out.alarm_hp;
      = "A-ALARMS".VALVES.err2.%X6;

      A "A-DBVALVES".ST3.SWORD_RISING.out.alarm_wp;
      = "A-ALARMS".VALVES.err2.%X8;

      CALL "A-TESTSCL"
      (  in_nr                       := 22 ,
         out                         := "A-DBVALVES".ST3.SWORD_RISING.test
      );

      A(;
      L "A-Doku_DB_OP".HMI.Manual_Functions;
      L 22;
      <>I;
      );
      R "A-DBVALVES".ST3.SWORD_RISING.test.fp_HP;
      R "A-DBVALVES".ST3.SWORD_RISING.test.fp_WP;
      R "A-DBVALVES".ST3.SWORD_RISING.test.fp_IDLE;

      O "A-DBVALVES".ST3.SWORD_RISING.interlock.hp_active;
      O "A-DBVALVES".ST3.SWORD_RISING.interlock.wp_active;
      O "A-DBVALVES".ST3.SWORD_RISING.interlock.idle_active;
      = "A-DBVALVES".io[22].interlock_vis;
NETWORK
TITLE = -

NETWORK
TITLE = [23] ST3 ZDERZAK - HP
//[23] ST3 BUMPER - HP
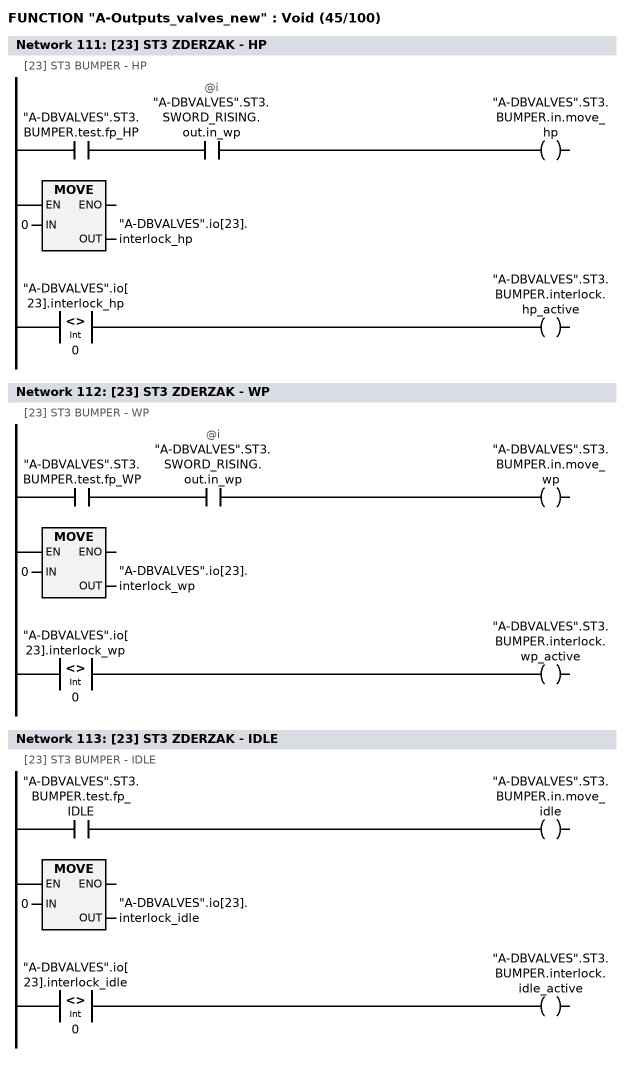
      O "A-DBVALVES".ST3.BUMPER.test.fp_HP;
//    O     "A-Flags".STATION.IN_HP_STEP
      A "A-DBVALVES".ST3.SWORD_RISING.out.in_wp;// @i
      = "A-DBVALVES".ST3.BUMPER.in.move_hp;

// Interlock hp
      L 0;
      T "A-DBVALVES".io[23].interlock_hp;

//{INTERLOCK_HP23}

      A(;
      L "A-DBVALVES".io[23].interlock_hp;
      L 0;
      <>I;
      );
      = "A-DBVALVES".ST3.BUMPER.interlock.hp_active;
NETWORK
TITLE = [23] ST3 ZDERZAK - WP
//[23] ST3 BUMPER - WP
      O "A-DBVALVES".ST3.BUMPER.test.fp_WP;
      A "A-DBVALVES".ST3.SWORD_RISING.out.in_wp;// @i
      = "A-DBVALVES".ST3.BUMPER.in.move_wp;

// Interlock wp
      L 0;
      T "A-DBVALVES".io[23].interlock_wp;

//{INTERLOCK_WP23}

      A(;
      L "A-DBVALVES".io[23].interlock_wp;
      L 0;
      <>I;
      );
      = "A-DBVALVES".ST3.BUMPER.interlock.wp_active;
NETWORK
TITLE = [23] ST3 ZDERZAK - IDLE
//[23] ST3 BUMPER - IDLE
      O "A-DBVALVES".ST3.BUMPER.test.fp_IDLE;
      = "A-DBVALVES".ST3.BUMPER.in.move_idle;

// Interlock idle
      L 0;
      T "A-DBVALVES".io[23].interlock_idle;

//{INTERLOCK_IDLE23}

      A(;
      L "A-DBVALVES".io[23].interlock_idle;
      L 0;
      <>I;
      );
      = "A-DBVALVES".ST3.BUMPER.interlock.idle_active;
NETWORK
TITLE = [23] ST3 ZDERZAK
//[23] ST3 BUMPER
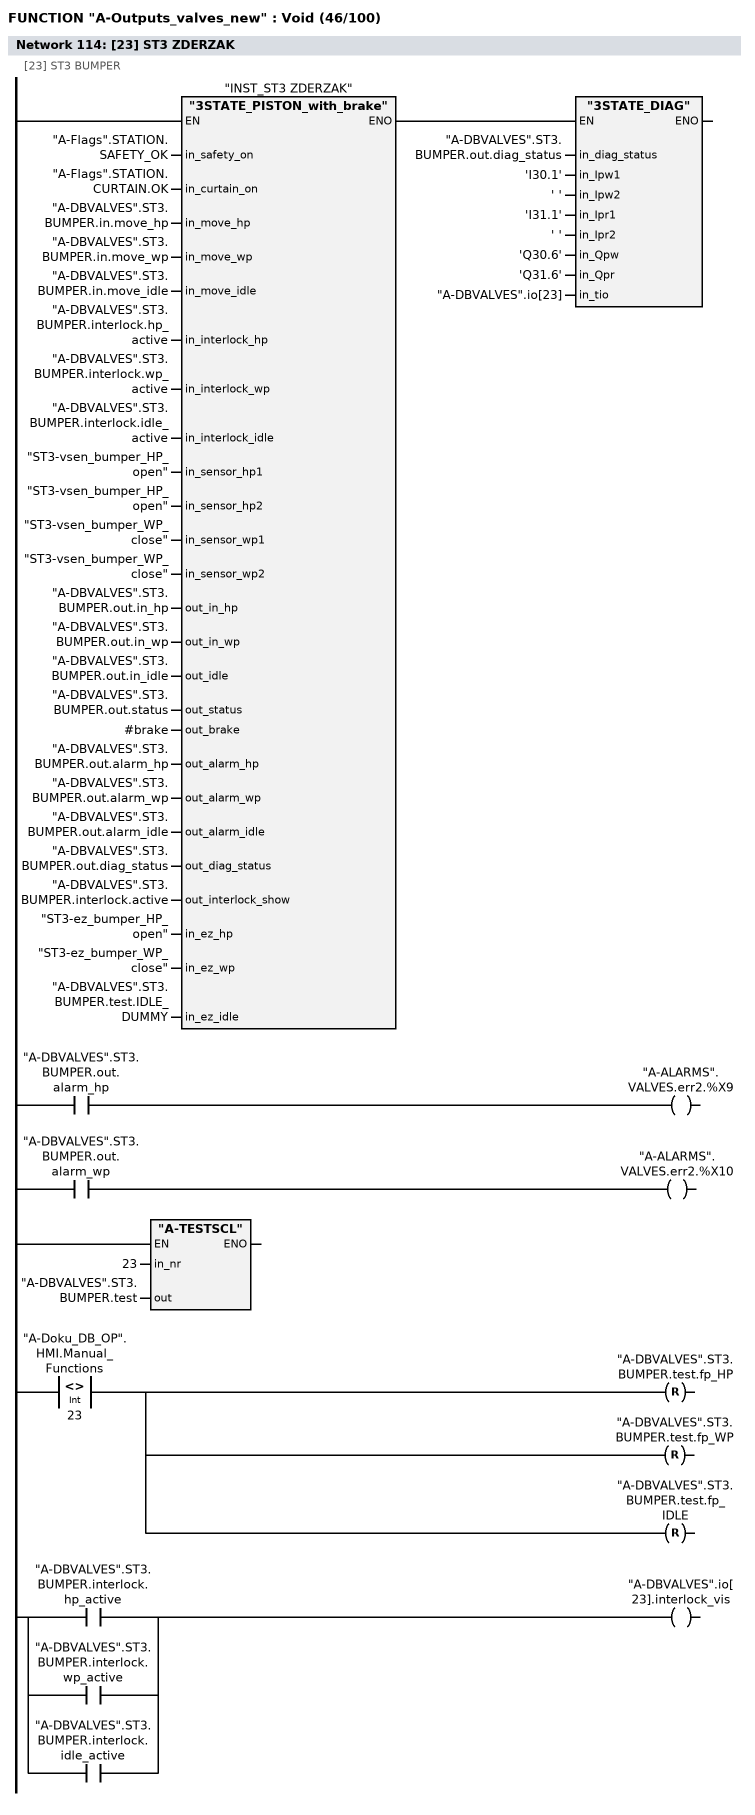
      CALL "3STATE_PISTON_with_brake", "INST_ST3 ZDERZAK"
      (  in_safety_on                := "A-Flags".STATION.SAFETY_OK ,
         in_curtain_on               := "A-Flags".STATION.CURTAIN.OK ,
         in_move_hp                  := "A-DBVALVES".ST3.BUMPER.in.move_hp ,
         in_move_wp                  := "A-DBVALVES".ST3.BUMPER.in.move_wp ,
         in_move_idle                := "A-DBVALVES".ST3.BUMPER.in.move_idle ,
         in_interlock_hp             := "A-DBVALVES".ST3.BUMPER.interlock.hp_active ,
         in_interlock_wp             := "A-DBVALVES".ST3.BUMPER.interlock.wp_active ,
         in_interlock_idle           := "A-DBVALVES".ST3.BUMPER.interlock.idle_active ,
         in_sensor_hp1               := "ST3-vsen_bumper_HP_open" ,
         in_sensor_hp2               := "ST3-vsen_bumper_HP_open" ,
         in_sensor_wp1               := "ST3-vsen_bumper_WP_close" ,
         in_sensor_wp2               := "ST3-vsen_bumper_WP_close" ,
         out_in_hp                   := "A-DBVALVES".ST3.BUMPER.out.in_hp ,
         out_in_wp                   := "A-DBVALVES".ST3.BUMPER.out.in_wp ,
         out_idle                    := "A-DBVALVES".ST3.BUMPER.out.in_idle ,
         out_status                  := "A-DBVALVES".ST3.BUMPER.out.status ,
         out_brake                   := #brake ,
         out_alarm_hp                := "A-DBVALVES".ST3.BUMPER.out.alarm_hp ,
         out_alarm_wp                := "A-DBVALVES".ST3.BUMPER.out.alarm_wp ,
         out_alarm_idle              := "A-DBVALVES".ST3.BUMPER.out.alarm_idle ,
         out_diag_status             := "A-DBVALVES".ST3.BUMPER.out.diag_status ,
         out_interlock_show          := "A-DBVALVES".ST3.BUMPER.interlock.active ,
         in_ez_hp                    := "ST3-ez_bumper_HP_open" ,
         in_ez_wp                    := "ST3-ez_bumper_WP_close" ,
         in_ez_idle                  := "A-DBVALVES".ST3.BUMPER.test.IDLE_DUMMY
      );

      CALL "3STATE_DIAG"
      (  in_diag_status              := "A-DBVALVES".ST3.BUMPER.out.diag_status ,
         in_Ipw1                     := 'I30.1' ,
         in_Ipw2                     := ' ' ,
         in_Ipr1                     := 'I31.1' ,
         in_Ipr2                     := ' ' ,
         in_Qpw                      := 'Q30.6' ,
         in_Qpr                      := 'Q31.6' ,
         in_tio                      := "A-DBVALVES".io[23]
      );

      A "A-DBVALVES".ST3.BUMPER.out.alarm_hp;
      = "A-ALARMS".VALVES.err2.%X9;

      A "A-DBVALVES".ST3.BUMPER.out.alarm_wp;
      = "A-ALARMS".VALVES.err2.%X10;

      CALL "A-TESTSCL"
      (  in_nr                       := 23 ,
         out                         := "A-DBVALVES".ST3.BUMPER.test
      );

      A(;
      L "A-Doku_DB_OP".HMI.Manual_Functions;
      L 23;
      <>I;
      );
      R "A-DBVALVES".ST3.BUMPER.test.fp_HP;
      R "A-DBVALVES".ST3.BUMPER.test.fp_WP;
      R "A-DBVALVES".ST3.BUMPER.test.fp_IDLE;

      O "A-DBVALVES".ST3.BUMPER.interlock.hp_active;
      O "A-DBVALVES".ST3.BUMPER.interlock.wp_active;
      O "A-DBVALVES".ST3.BUMPER.interlock.idle_active;
      = "A-DBVALVES".io[23].interlock_vis;
NETWORK
TITLE = -

NETWORK
TITLE = [24] ST3 MIECZ - HP
//[24] ST3 SWORD - HP
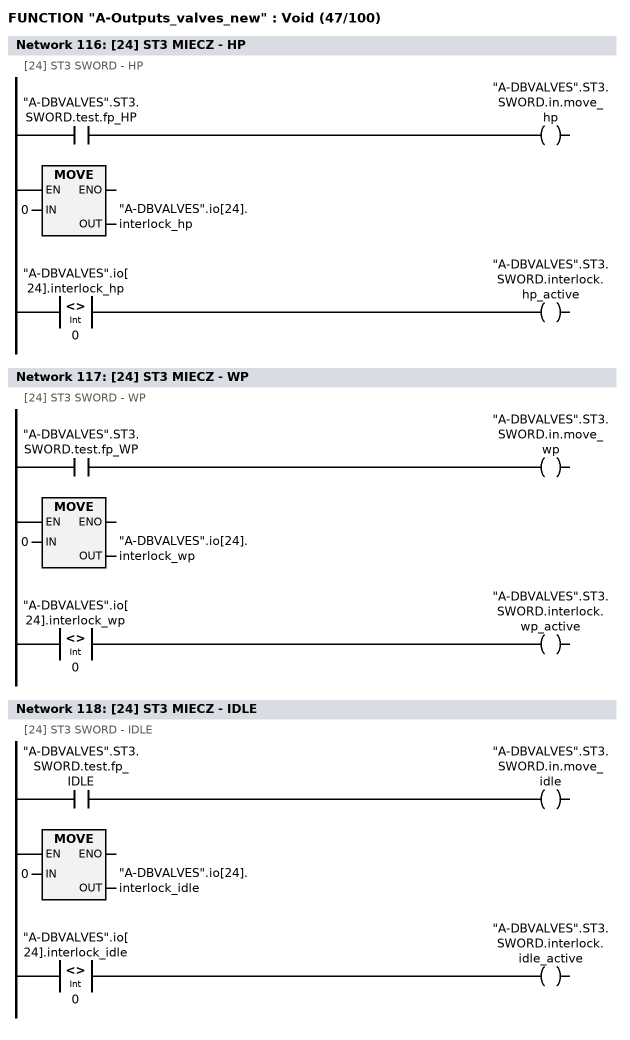
      O "A-DBVALVES".ST3.SWORD.test.fp_HP;
//    O     "A-Flags".STATION.IN_HP_STEP
      = "A-DBVALVES".ST3.SWORD.in.move_hp;

// Interlock hp
      L 0;
      T "A-DBVALVES".io[24].interlock_hp;

//{INTERLOCK_HP24}

      A(;
      L "A-DBVALVES".io[24].interlock_hp;
      L 0;
      <>I;
      );
      = "A-DBVALVES".ST3.SWORD.interlock.hp_active;
NETWORK
TITLE = [24] ST3 MIECZ - WP
//[24] ST3 SWORD - WP
      O "A-DBVALVES".ST3.SWORD.test.fp_WP;
      = "A-DBVALVES".ST3.SWORD.in.move_wp;

// Interlock wp
      L 0;
      T "A-DBVALVES".io[24].interlock_wp;

//{INTERLOCK_WP24}

      A(;
      L "A-DBVALVES".io[24].interlock_wp;
      L 0;
      <>I;
      );
      = "A-DBVALVES".ST3.SWORD.interlock.wp_active;
NETWORK
TITLE = [24] ST3 MIECZ - IDLE
//[24] ST3 SWORD - IDLE
      O "A-DBVALVES".ST3.SWORD.test.fp_IDLE;
      = "A-DBVALVES".ST3.SWORD.in.move_idle;

// Interlock idle
      L 0;
      T "A-DBVALVES".io[24].interlock_idle;

//{INTERLOCK_IDLE24}

      A(;
      L "A-DBVALVES".io[24].interlock_idle;
      L 0;
      <>I;
      );
      = "A-DBVALVES".ST3.SWORD.interlock.idle_active;
NETWORK
TITLE = [24] ST3 MIECZ
//[24] ST3 SWORD
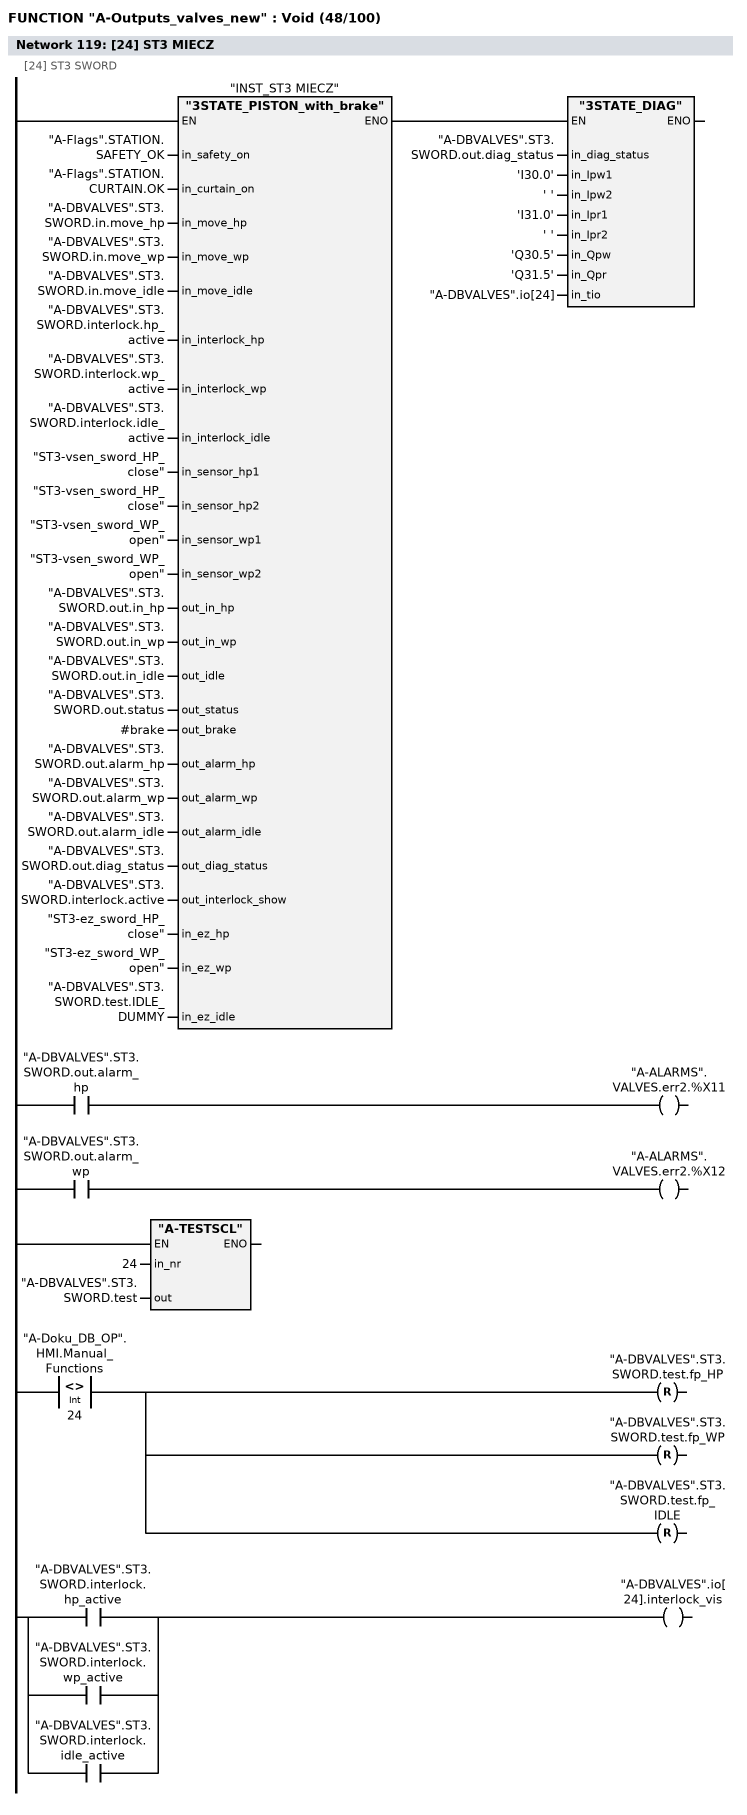
      CALL "3STATE_PISTON_with_brake", "INST_ST3 MIECZ"
      (  in_safety_on                := "A-Flags".STATION.SAFETY_OK ,
         in_curtain_on               := "A-Flags".STATION.CURTAIN.OK ,
         in_move_hp                  := "A-DBVALVES".ST3.SWORD.in.move_hp ,
         in_move_wp                  := "A-DBVALVES".ST3.SWORD.in.move_wp ,
         in_move_idle                := "A-DBVALVES".ST3.SWORD.in.move_idle ,
         in_interlock_hp             := "A-DBVALVES".ST3.SWORD.interlock.hp_active ,
         in_interlock_wp             := "A-DBVALVES".ST3.SWORD.interlock.wp_active ,
         in_interlock_idle           := "A-DBVALVES".ST3.SWORD.interlock.idle_active ,
         in_sensor_hp1               := "ST3-vsen_sword_HP_close" ,
         in_sensor_hp2               := "ST3-vsen_sword_HP_close" ,
         in_sensor_wp1               := "ST3-vsen_sword_WP_open" ,
         in_sensor_wp2               := "ST3-vsen_sword_WP_open" ,
         out_in_hp                   := "A-DBVALVES".ST3.SWORD.out.in_hp ,
         out_in_wp                   := "A-DBVALVES".ST3.SWORD.out.in_wp ,
         out_idle                    := "A-DBVALVES".ST3.SWORD.out.in_idle ,
         out_status                  := "A-DBVALVES".ST3.SWORD.out.status ,
         out_brake                   := #brake ,
         out_alarm_hp                := "A-DBVALVES".ST3.SWORD.out.alarm_hp ,
         out_alarm_wp                := "A-DBVALVES".ST3.SWORD.out.alarm_wp ,
         out_alarm_idle              := "A-DBVALVES".ST3.SWORD.out.alarm_idle ,
         out_diag_status             := "A-DBVALVES".ST3.SWORD.out.diag_status ,
         out_interlock_show          := "A-DBVALVES".ST3.SWORD.interlock.active ,
         in_ez_hp                    := "ST3-ez_sword_HP_close" ,
         in_ez_wp                    := "ST3-ez_sword_WP_open" ,
         in_ez_idle                  := "A-DBVALVES".ST3.SWORD.test.IDLE_DUMMY
      );

      CALL "3STATE_DIAG"
      (  in_diag_status              := "A-DBVALVES".ST3.SWORD.out.diag_status ,
         in_Ipw1                     := 'I30.0' ,
         in_Ipw2                     := ' ' ,
         in_Ipr1                     := 'I31.0' ,
         in_Ipr2                     := ' ' ,
         in_Qpw                      := 'Q30.5' ,
         in_Qpr                      := 'Q31.5' ,
         in_tio                      := "A-DBVALVES".io[24]
      );

      A "A-DBVALVES".ST3.SWORD.out.alarm_hp;
      = "A-ALARMS".VALVES.err2.%X11;

      A "A-DBVALVES".ST3.SWORD.out.alarm_wp;
      = "A-ALARMS".VALVES.err2.%X12;

      CALL "A-TESTSCL"
      (  in_nr                       := 24 ,
         out                         := "A-DBVALVES".ST3.SWORD.test
      );

      A(;
      L "A-Doku_DB_OP".HMI.Manual_Functions;
      L 24;
      <>I;
      );
      R "A-DBVALVES".ST3.SWORD.test.fp_HP;
      R "A-DBVALVES".ST3.SWORD.test.fp_WP;
      R "A-DBVALVES".ST3.SWORD.test.fp_IDLE;

      O "A-DBVALVES".ST3.SWORD.interlock.hp_active;
      O "A-DBVALVES".ST3.SWORD.interlock.wp_active;
      O "A-DBVALVES".ST3.SWORD.interlock.idle_active;
      = "A-DBVALVES".io[24].interlock_vis;
NETWORK
TITLE = -

NETWORK
TITLE = [25] ST4 MIECZ_PODNOSZENIE - HP
//[25] ST4 SWORD_RISING - HP
